// TIA Portal project "s7netcsharp_V16" (V16)

(* hardware
DEVICE "S7300/ET200M station_1"  S7-300 station
   slot 0: "Rail_0"  Rail  6ES7 390-1***0-0AA0
   slot 2: "PLC_1"  CPU 315-2 PN/DP  6ES7 315-2EH14-0AB0  V3.2
      slot 2: "PROFINET interface_1"  PN-IO
         slot 1: "Port_1"  Port
         slot 2: "Port_2"  Port
*)

// ===== PLC "PLC_1"  CPU 315-2 PN/DP =====

VAR_GLOBAL   // PLC tag table "Default tag table"
   "Tag_1" AT %M10.0 : Bool;
   "Tag_2" AT %M10.1 : Bool;
   "Tag_3" AT %M10.2 : Bool;
   "Tag_4" AT %M10.3 : Bool;
   "Tag_5" AT %MW12 : Word;
   "Tag_6" AT %M10.6 : Bool;
   "Tag_7" AT %M10.7 : Bool;
   "Tag_8" AT %MW14 : Word;
   "Tag_9" AT %M11.0 : Bool;
   "Tag_10" AT %M11.1 : Bool;
   "Tag_11" AT %M11.2 : Bool;
   "Tag_12" AT %M11.3 : Bool;
   "Tag_13" AT %M11.4 : Bool;
   "Tag_14" AT %M11.5 : Bool;
   "Tag_15" AT %MW16 : Word;
   "Tag_16" AT %M11.6 : Bool;
   "Tag_17" AT %M20.1 : Bool;
   "Tag_18" AT %M20.2 : Bool;
   "Tag_19" AT %MW22 : Word;
   "Tag_20" AT %M20.4 : Bool;
   "Tag_21" AT %M20.3 : Bool;
   "Tag_22" AT %M20.0 : Bool;
   "Tag_23" AT %M10.4 : Bool;
   "Tag_24" AT %M21.0 : Bool;
   "Tag_25" AT %M21.1 : Bool;
   "AlwaysFalse" AT %M1.0 : Bool;
   "AlwaysTrue" AT %M1.1 : Bool;
   "Tag_26" AT %M0.0 : Bool;
   "Tag_27" AT %M0.1 : Bool;
   "Tag_28" AT %M0.2 : Bool;
   "Tag_29" AT %M0.3 : Bool;
   "Tag_30" AT %M0.4 : Bool;
   "Clock_1Hz" AT %M0.5 : Bool;
   "Time" AT %MD24 : Time;
   "TimeInt" AT %MW28 : Int;
   "pH" AT %MD30 : Real;
END_VAR

DATA_BLOCK "Test"   // DB2
{ S7_Optimized_Access := 'FALSE' }
VERSION : 0.1
   VAR
      Test : Real;
      TestInt : Int;
   END_VAR
BEGIN
END_DATA_BLOCK

// folder: Calculation

DATA_BLOCK "FB_Scale_LI_2"   // DB6
{ S7_Optimized_Access := 'FALSE' }
VERSION : 0.1
// stored: InstanceOfName FB_Scale
"FB_Scale"
BEGIN
END_DATA_BLOCK

DATA_BLOCK "DB_CalculateFlow_FI_1"   // DB13
{ S7_Optimized_Access := 'FALSE' }
VERSION : 0.1
// stored: InstanceOfName FB_CalculateFlow
"FB_CalculateFlow"
BEGIN
END_DATA_BLOCK

DATA_BLOCK "DB_CalculateFlow_FI_2"   // DB14
{ S7_Optimized_Access := 'FALSE' }
VERSION : 0.1
// stored: InstanceOfName FB_CalculateFlow
"FB_CalculateFlow"
BEGIN
END_DATA_BLOCK

DATA_BLOCK "DB_FillingTankT1"   // DB16
{ S7_Optimized_Access := 'FALSE' }
VERSION : 0.1
// stored: InstanceOfName FB_FillingTankT1
"FB_FillingTankT1"
BEGIN
END_DATA_BLOCK

DATA_BLOCK "DB_FillingTankT2"   // DB17
{ S7_Optimized_Access := 'FALSE' }
VERSION : 0.1
// stored: InstanceOfName FB_FillingTankT2
"FB_FillingTankT2"
BEGIN
END_DATA_BLOCK

DATA_BLOCK "FB_Scale_LI_1"   // DB23
{ S7_Optimized_Access := 'FALSE' }
VERSION : 0.1
// stored: InstanceOfName FB_Scale
"FB_Scale"
BEGIN
END_DATA_BLOCK

DATA_BLOCK "DB_PhCalculation"   // DB25
{ S7_Optimized_Access := 'FALSE' }
VERSION : 0.1
// stored: InstanceOfName FB_PhCalculation
"FB_PhCalculation"
BEGIN
END_DATA_BLOCK

DATA_BLOCK "DB_EmptyingCT"   // DB26
{ S7_Optimized_Access := 'FALSE' }
VERSION : 0.1
// stored: InstanceOfName FB_EmptyingCT
"FB_EmptyingCT"
BEGIN
END_DATA_BLOCK

// folder: Measuring Points

DATA_BLOCK "Digital sensors"   // DB7
{ S7_Optimized_Access := 'FALSE' }
VERSION : 0.1
   VAR
      LSHH_T1 : Bool;   // Very high level in Tank 1
      LSLL_T1 : Bool;   // Very low level in Tank 1
      LSHH_T2 : Bool;   // Very high level in Tank 3
      LSLL_T2 : Bool;   // Very low level in Tank 3
      LSH_CT : Bool;   // High level in Chemicals Tank 1
      LSL_CT : Bool;   // Low level in Chemicals Tank 1
   END_VAR
BEGIN
END_DATA_BLOCK

// folder: Measuring Points/Analogs

DATA_BLOCK "DB_Analog_LI_1"   // DB4
{ S7_Optimized_Access := 'FALSE' }
VERSION : 0.1
// stored: InstanceOfName FB_Analog
"FB_Analog"
BEGIN
END_DATA_BLOCK

DATA_BLOCK "DB_Analog_FI_1"   // DB19
{ S7_Optimized_Access := 'FALSE' }
VERSION : 0.1
// stored: InstanceOfName FB_Analog
"FB_Analog"
BEGIN
END_DATA_BLOCK

DATA_BLOCK "DB_Analog_LI_2"   // DB20
{ S7_Optimized_Access := 'FALSE' }
VERSION : 0.1
// stored: InstanceOfName FB_Analog
"FB_Analog"
BEGIN
END_DATA_BLOCK

DATA_BLOCK "DB_Analog_AI_1"   // DB21
{ S7_Optimized_Access := 'FALSE' }
VERSION : 0.1
// stored: InstanceOfName FB_Analog
"FB_Analog"
BEGIN
END_DATA_BLOCK

DATA_BLOCK "DB_Analog_FI_2"   // DB22
{ S7_Optimized_Access := 'FALSE' }
VERSION : 0.1
// stored: InstanceOfName FB_Analog
"FB_Analog"
BEGIN
END_DATA_BLOCK

// folder: Measuring Points/Measuring Transducers

DATA_BLOCK "DB_LI_1"   // DB1
{ S7_Optimized_Access := 'FALSE' }
VERSION : 0.1
// stored: InstanceOfName FB_MeasuringTransducer
"FB_MeasuringTransducer"
BEGIN
END_DATA_BLOCK

DATA_BLOCK "DB_FI_1"   // DB5
{ S7_Optimized_Access := 'FALSE' }
VERSION : 0.1
// stored: InstanceOfName FB_MeasuringTransducer
"FB_MeasuringTransducer"
BEGIN
END_DATA_BLOCK

DATA_BLOCK "DB_LI_2"   // DB28
{ S7_Optimized_Access := 'FALSE' }
VERSION : 0.1
// stored: InstanceOfName FB_MeasuringTransducer
"FB_MeasuringTransducer"
BEGIN
END_DATA_BLOCK

DATA_BLOCK "DB_AI_1"   // DB29
{ S7_Optimized_Access := 'FALSE' }
VERSION : 0.1
// stored: InstanceOfName FB_MeasuringTransducer
"FB_MeasuringTransducer"
BEGIN
END_DATA_BLOCK

DATA_BLOCK "DB_FI_2"   // DB30
{ S7_Optimized_Access := 'FALSE' }
VERSION : 0.1
// stored: InstanceOfName FB_MeasuringTransducer
"FB_MeasuringTransducer"
BEGIN
END_DATA_BLOCK

// folder: Program files

DATA_BLOCK "DB_FILL_T1"   // DB12
{ S7_Optimized_Access := 'FALSE' }
VERSION : 0.1
   VAR
      START : Bool;   // Start signal from SCADA
      SET_START : Bool;   // Set start signal
      STOP : Bool;   // Stop signal from SCADA
      SET_STOP : Bool;   // Set stop signal
      UV_1_OPEN : Bool;   // Open valve UV_1
      STATE : Int;   // 0 - Stop, 1 - Filling T1, 2 - No conditions to run
   END_VAR
BEGIN
END_DATA_BLOCK

DATA_BLOCK "DB_TRANSFER_TO_T2"   // DB18
{ S7_Optimized_Access := 'FALSE' }
VERSION : 0.1
   VAR
      START : Bool;   // Start signal from SCADA
      SET_START : Bool;   // Set start signal
      STOP : Bool;   // Stop signal from SCADA
      SET_STOP : Bool;   // Set stop signal
      Spare : Bool;   // Spare
      P1_START : Bool;   // Start signal for Pump P1
      UV_2_OPEN : Bool;   // Open valve UV_2
      SetPhVal : Bool;   // Set random ph value signal
      LI_2_SP : Real := 7000.0;   // Setpoint for Tank T2 filling level
      AI_1_SetVal : Real;   // Random Value of Ph in Tank T3
      STATE : Int;   // 0 - Stop, 1 - Transfer to T2, 2 - Adding chemicals, 3 - No conditions to run
      P1_SP : Real;   // Pump P1 Speed Setpoint
   END_VAR
BEGIN
END_DATA_BLOCK

DATA_BLOCK "DB_DOSE_CHEMICALS"   // DB24
{ S7_Optimized_Access := 'FALSE' }
VERSION : 0.1
   VAR
      START : Bool;   // Start signal from SCADA
      SET_START : Bool;   // Set start signal
      STOP : Bool;   // Stop signal from SCADA
      SET_STOP : Bool;   // Set stop signal
      P3_START : Bool;
      STATE : Int;   // 0 - Stop, 1 - Adding Chemicals, 2 - No conditions to run
   END_VAR
BEGIN
END_DATA_BLOCK

DATA_BLOCK "DB_EMPTYING_T2"   // DB27
{ S7_Optimized_Access := 'FALSE' }
VERSION : 0.1
   VAR
      START : Bool;   // Start signal from SCADA
      SET_START : Bool;   // Set start signal
      STOP : Bool;   // Stop signal from SCADA
      SET_STOP : Bool;   // Set stop signal
      P2_START : Bool;   // Start signal for Pump P2
      Spare : Bool;
      Spare_1 : Bool;
      Spare_2 : Bool;
      State : Int;   // 0 - stop, 1 - Emptying, 3 - No conditions to run
      P2_SP : Real;   // Pump P2 Speed Setpoint
   END_VAR
BEGIN
END_DATA_BLOCK

// folder: Pumps

DATA_BLOCK "DB_Pump_P1"   // DB8
{ S7_Optimized_Access := 'FALSE' }
VERSION : 0.1
// stored: InstanceOfName FB_MotorControl
"FB_MotorControl"
BEGIN
END_DATA_BLOCK

DATA_BLOCK "DB_Pump_P2"   // DB9
{ S7_Optimized_Access := 'FALSE' }
VERSION : 0.1
// stored: InstanceOfName FB_MotorControl
"FB_MotorControl"
BEGIN
END_DATA_BLOCK

DATA_BLOCK "DB_Pump_P3"   // DB15
{ S7_Optimized_Access := 'FALSE' }
VERSION : 0.1
// stored: InstanceOfName FB_MotorControl
"FB_MotorControl"
BEGIN
END_DATA_BLOCK

// folder: Valves

DATA_BLOCK "DB_UV_1"   // DB10
{ S7_Optimized_Access := 'FALSE' }
VERSION : 0.1
// stored: InstanceOfName FB_Valve
"FB_Valve"
BEGIN
END_DATA_BLOCK

DATA_BLOCK "DB_UV_2"   // DB11
{ S7_Optimized_Access := 'FALSE' }
VERSION : 0.1
// stored: InstanceOfName FB_Valve
"FB_Valve"
BEGIN
END_DATA_BLOCK

// folder: (top level)

FUNCTION_BLOCK "FB_MeasuringTransducer"   // FB1, SCL
{ S7_Optimized_Access := 'FALSE' }
VERSION : 0.1
   VAR_INPUT
      X : Real;   // Input value (Final respond transducer value
      T1 : Time;   // Main constant transducer value
      T2 : Time;   // Second constant transducer value
      Ts : Time;   // Sampling time
      K : Real;   // Gain
   END_VAR
   VAR_OUTPUT
      Y : Real;   // Output value
   END_VAR
   VAR
      Yn1 : Real;
      Yn2 : Real;
      T_Sampling : Real;
      T1_Temp : Real;
      T2_Temp : Real;
   END_VAR
BEGIN
   // Input time conversion
   #T_Sampling := (DINT_TO_REAL(TIME_TO_DINT(#Ts))) / 1000.0;
   #T1_Temp := (DINT_TO_REAL(TIME_TO_DINT(#T1))) / 1000.0;
   #T2_Temp := (DINT_TO_REAL(TIME_TO_DINT(#T2))) / 1000.0;

   // ***************************************************
   // Second order measuring transducer Euler's equation
   // For more details go to Readme.txt file
   // ***************************************************

   #Y := ((#K * (#T_Sampling * #T_Sampling) * #X) + ((#T_Sampling
   * #T1_Temp + 2 * #T1_Temp * #T2_Temp + #T_Sampling * #T2_Temp) *
   #Yn1) - ((#T1_Temp * #T2_Temp) * #Yn2)) / ((#T_Sampling *
   #T_Sampling) + #T_Sampling * #T2_Temp + #T_Sampling * #T1_Temp +
   #T1_Temp * #T2_Temp);

   #Yn2 := #Yn1;
   #Yn1 := #Y;
END_FUNCTION_BLOCK

FUNCTION_BLOCK "FB_MotorControl"   // FB2, SCL
{ S7_Optimized_Access := 'FALSE' }
VERSION : 0.1
   VAR_INPUT
      START : Bool;   // Start in auto mode
      BLOCKADE : Bool;
      TRIGGER : Bool;   // Time trigger for running time
      SP_IN : Real;   // Setpoint [%]
   END_VAR
   VAR_OUTPUT
      RUNNING : Bool;
      FAULT : Bool;
      ERROR_CODE : Int;
      STATE : Int;   // 0 - stop, 1 - starting up, 2 - run, 3 - stopping, 4 - blockade active, 5 - fault
      PV : Real;
   END_VAR
   VAR
      MODE : Bool := false;   // 0 - auto, 1 - manual
      SCADA : Struct   // Signals from/to Scada
         START : Bool;   // Start signal from Scada
         STOP : Bool;   // Stop signal from Scada
         AUTO : Bool := false;   // Auto mode signal from Scada
         MANUAL : Bool;   // Manual mode signal from Scada
         BLOCKADE : Bool;   // 0 - blockade unactive, 1 - blockade active
         FAULT : Bool;   // Motor fault info to Scada
         RUN_H : Int;   // Running time - hours
         RUN_MIN : Int;   // Running time - minutes
         RUN_S : Int;   // Running time - seconds
         RESET_TIME : Bool;   // Reset running time
         MODE : Bool;   // 0 - auto, 1 - manual (Scada)
         STATE : Int;   // 0 - stop, 1 - starting up, 2 - running, 3 - stopping, 4 - blockade active, 5 - fault
         SP : Real;   // Setpoint value [%]
         PV : Real;
      END_STRUCT;
      Yn1 : Real;
      Yn2 : Real;
      T_Sampling : Real;
      T1_Temp : Real;
      T2_Temp : Real;
      SP : Real;
      SignalOld : Bool;
   END_VAR
   VAR_TEMP
      Edge : Bool;
   END_VAR
   VAR CONSTANT
      T1 : Time := T#1s;   // Main constant transducer value
      T2 : Time := T#500ms;   // Second constant transducer value
      Ts : Time := T#100ms;   // Sampling time
      K : Real := 1.0;   // Gain
   END_VAR
BEGIN
   #SCADA.BLOCKADE := #BLOCKADE;
   #SCADA.FAULT := #FAULT;
   #SCADA.STATE := #STATE;

   // Input time conversion
   #T_Sampling := (DINT_TO_REAL(TIME_TO_DINT(#Ts))) / 1000.0;
   #T1_Temp := (DINT_TO_REAL(TIME_TO_DINT(#T1))) / 1000.0;
   #T2_Temp := (DINT_TO_REAL(TIME_TO_DINT(#T2))) / 1000.0;

   // Positive edge detection
   #Edge := #TRIGGER AND NOT #SignalOld;
   #SignalOld := #TRIGGER;

   // Blockade
   IF (#BLOCKADE) THEN
       #ERROR_CODE := 1;
       #START := FALSE;
       #SCADA.START := FALSE;
       #SCADA.STOP := TRUE;
       #RUNNING := FALSE;
       #FAULT := TRUE;
       #SP := 0;
       #STATE := 4;
   END_IF;

   // Manual and auto mode set
   IF (#SCADA.MANUAL) THEN
       #MODE := TRUE;
   ELSIF (#SCADA.AUTO) THEN
       #MODE := FALSE;
   END_IF;

   // Main program
   IF (#BLOCKADE = FALSE) THEN
       #FAULT := FALSE;
       IF (#MODE = FALSE AND #START = TRUE) THEN
           #RUNNING := TRUE;
           #SP := #SP_IN;

           //Status change - starting up/run
           IF (#SP * 0.90 > #PV) THEN
               #STATE := 1;
           ELSIF (#SP * 0.90 < #PV) THEN
               #STATE := 2;
           END_IF;

       ELSIF (#MODE = FALSE AND #START = FALSE) THEN
           #RUNNING := FALSE;
           #SP := 0.0;
           //Status change - stopping/stop
           IF (0.05 < #PV) THEN
               #STATE := 3;
           ELSIF (0.05 > #PV) THEN
               #STATE := 4;
           END_IF;

       ELSIF(#MODE = TRUE AND #SCADA.START = TRUE) THEN
           #RUNNING := TRUE;
           #SP := #SCADA.SP;
           //Status change - starting up/runn
           IF (#SP * 0.90 > #PV) THEN
               #STATE := 1;
           ELSIF (#SP * 0.90 < #PV) THEN
               #STATE := 2;
           END_IF;

       ELSIF (#MODE = TRUE AND #SCADA.START = FALSE) THEN
           #RUNNING := FALSE;
           #SP := 0.0;
           //Status change - stopping/stop
           IF (0.05 < #PV) THEN
               #STATE := 3;
           ELSIF (0.05 > #PV) THEN
               #STATE := 4;
           END_IF;

       END_IF;
   END_IF;

   // Euler's second order equation for simulate acceleration and slowing down  
   #PV := ((#K * (#T_Sampling * #T_Sampling) * #SP) + ((#T_Sampling
   * #T1_Temp + 2 * #T1_Temp * #T2_Temp + #T_Sampling * #T2_Temp) *
   #Yn1) - ((#T1_Temp * #T2_Temp) * #Yn2)) / ((#T_Sampling *
   #T_Sampling) + #T_Sampling * #T2_Temp + #T_Sampling * #T1_Temp +
   #T1_Temp * #T2_Temp);
   #Yn2 := #Yn1;
   #Yn1 := #PV;

   // Running time
   IF (#RUNNING AND #Edge) THEN
       #SCADA.RUN_S := #SCADA.RUN_S+1;
       IF (#SCADA.RUN_S = 60) THEN
           #SCADA.RUN_S := 0;
           #SCADA.RUN_MIN := #SCADA.RUN_MIN+1;
       END_IF;

       IF (#SCADA.RUN_MIN = 60) THEN
           #SCADA.RUN_MIN := 0;
           #SCADA.RUN_H := #SCADA.RUN_H+1;
       END_IF;

   END_IF;

   // Reset running time
   IF (#SCADA.RESET_TIME) THEN
       #SCADA.RUN_S := 0;
       #SCADA.RUN_MIN := 0;
       #SCADA.RUN_H := 0;
   END_IF;

   // 
   // STATUS CODES
   // 1: Blockade active
   //
END_FUNCTION_BLOCK

FUNCTION_BLOCK "FB_Valve"   // FB3, SCL
{ S7_Optimized_Access := 'FALSE' }
VERSION : 0.1
   VAR_INPUT
      "OPEN/CLOSE" : Bool;   // 0 - Close, 1 - Open
      BLOCKADE : Bool;
      DETECT_TIME : Int;   // Time of Inefficient open / close detection error [s]
   END_VAR
   VAR_OUTPUT
      STATE : Int;   // 0 - Closed, 1 - Closing, 2 - Open, 3 - Opening, 4 - Fault
      FAULT : Bool;
      ERROR_CODE : Int;
      OUT : Bool;   // 0 - Close, 1 - Open
      CLOSE_LIMIT : Bool;   // Closing limit
      OPEN_LIMIT : Bool;   // Opening limit
   END_VAR
   VAR
      SCADA : Struct
         OPEN : Bool;   // Open valve singal from scada
         CLOSE : Bool;   // Close valve singal from scada
         AUTO : Bool;   // Auto mode signal from scada
         MANUAL : Bool;   // Manual mode signal from scada
         FAULT : Bool;   // Valve fault
         BLOCKADE : Bool;   // 1 - Blockade active
         AM : Bool;   // 0 - Auto, 1 - Manual
         OPEN_CLOSE : Bool;   // 0 - Closing, 1 - Opening
         STATE : Int;   // 0 - Closed, 1 - Closing, 2 - Open, 3 - Opening
      END_STRUCT;
      SignalOld : Bool;
      OpenDetTime : Int;
      CloseDetTime : Int;
   END_VAR
   VAR_TEMP
      EDGE : Bool;
   END_VAR
BEGIN
   #SCADA.STATE := #STATE;
   #SCADA.FAULT := #FAULT;
   #SCADA.BLOCKADE := #BLOCKADE;
   // Positive edge detection
   #EDGE := "Clock_1Hz" AND NOT #SignalOld;
   #SignalOld := "Clock_1Hz";

   // Open / Close from scada
   IF (#SCADA.OPEN) THEN
       #SCADA.OPEN_CLOSE := TRUE;
       #SCADA.OPEN := FALSE;
   ELSIF (#SCADA.CLOSE) THEN
       #SCADA.OPEN_CLOSE := FALSE;
       #SCADA.CLOSE := FALSE;
   END_IF;

   // Auto / Manual from scada
   IF (#SCADA.MANUAL) THEN
       #SCADA.AM := TRUE;
       #SCADA.MANUAL := FALSE;
   ELSIF (#SCADA.AUTO) THEN
       #SCADA.AM := FALSE;
       #SCADA.AUTO := FALSE;
   END_IF;

   IF (#BLOCKADE) THEN
       #FAULT := TRUE;
       #OUT := FALSE;
       #ERROR_CODE := 1;
       #OpenDetTime := 0;

       //Close valve when blockade is on
       IF (#EDGE AND #CloseDetTime <> #DETECT_TIME) THEN
           #CloseDetTime := #CloseDetTime + 1;
           #STATE := 1;

           IF (#CloseDetTime = #DETECT_TIME) THEN
               #OUT := TRUE;
               #STATE := 0;
               #OPEN_LIMIT := FALSE;
               #CLOSE_LIMIT := TRUE;
           END_IF;

       END_IF;

   ELSIF (#BLOCKADE = FALSE) THEN
       #FAULT := FALSE;
       // Manual Mode
       IF (#SCADA.AM) THEN
           // Opening the valve
           IF (#SCADA.OPEN_CLOSE) THEN
               #CloseDetTime := 0;
               IF (#EDGE AND #OpenDetTime <> #DETECT_TIME) THEN
                   #OpenDetTime := #OpenDetTime + 1;
                   #STATE := 3;

                   IF (#OpenDetTime = #DETECT_TIME) THEN
                       #OUT := TRUE;
                       #STATE := 2;
                       #CLOSE_LIMIT := FALSE;
                       #OPEN_LIMIT := TRUE;
                   END_IF;

               END_IF;
           // Closing valve
           ELSIF (#SCADA.OPEN_CLOSE=FALSE) THEN
               #OpenDetTime := 0;
               IF (#EDGE AND #CloseDetTime <> #DETECT_TIME) THEN
                   #CloseDetTime := #CloseDetTime + 1;
                   #STATE := 1;

                   IF (#CloseDetTime = #DETECT_TIME) THEN
                       #OUT := TRUE;
                       #STATE := 0;
                       #OPEN_LIMIT := FALSE;
                       #CLOSE_LIMIT := TRUE;
                   END_IF;

               END_IF;
           END_IF;
       // Automatic mode    
       ELSIF (#SCADA.AM = FALSE) THEN
           // Opening the valve
           IF (#"OPEN/CLOSE") THEN
               #CloseDetTime := 0;
               IF (#EDGE AND #OpenDetTime <> #DETECT_TIME) THEN
                   #OpenDetTime := #OpenDetTime + 1;
                   #STATE := 3;

                   IF (#OpenDetTime = #DETECT_TIME) THEN
                       #OUT := TRUE;
                       #STATE := 2;
                       #CLOSE_LIMIT := FALSE;
                       #OPEN_LIMIT := TRUE;
                   END_IF;

               END_IF;
           // Closing valve    
           ELSIF (#"OPEN/CLOSE" = FALSE) THEN
               #OpenDetTime := 0;
               IF (#EDGE AND #CloseDetTime <> #DETECT_TIME) THEN
                   #CloseDetTime := #CloseDetTime + 1;
                   #STATE := 1;

                   IF (#CloseDetTime = #DETECT_TIME) THEN
                       #OUT := TRUE;
                       #STATE := 0;
                       #OPEN_LIMIT := FALSE;
                       #CLOSE_LIMIT := TRUE;
                   END_IF;

               END_IF;
           END_IF;

       END_IF;

   END_IF;
END_FUNCTION_BLOCK

FUNCTION_BLOCK "FB_Scale"   // FB7, SCL
{ S7_Optimized_Access := 'FALSE' }
VERSION : 0.1
   VAR_INPUT
      VALUE : Real;
      HI_RANGE : Real;
   END_VAR
   VAR_OUTPUT
      OUT_PRC : Real;
   END_VAR
BEGIN
   // Scale input value to percent

   #OUT_PRC := DINT_TO_REAL(ROUND(((#VALUE * 100.0) / #HI_RANGE) *100.0))/100.0;
END_FUNCTION_BLOCK

FUNCTION_BLOCK "FB_RandomPhGenerator"   // FB10, SCL
{ S7_Optimized_Access := 'FALSE' }
VERSION : 0.1
   VAR_INPUT
      LowRange : Real;   // Minimum input ph value ( 0 - min)
      HghRange : Real;   // Maximum input ph value (10 - max)
   END_VAR
   VAR_OUTPUT
      Value : Real;
      Error : Bool;   // Wrong input value (1-10ph)
   END_VAR
   VAR
      "Time" : Date_And_Time;
      Seconds : Int;
   END_VAR
   VAR_TEMP
      RetVal : Int;
   END_VAR
BEGIN
   #RetVal:=RD_SYS_T(OUT => #Time);
END_FUNCTION_BLOCK

FUNCTION_BLOCK "FB_Analog"   // FB11, SCL
{ S7_Optimized_Access := 'FALSE' }
VERSION : 0.1
   VAR_INPUT
      Value : Real;   // Measured Value
      HHI : Bool;   // Very high level of measured value (Alarm)
      HI : Bool;   // High level of measured value (Warning)
      LO : Bool;   // Low level of measured value (Warning)
      LLO : Bool;   // Very low level of measured value (Alarm)
      HHI_SP : Real;   // Setpoint for very high level detection
      HI_SP : Real;   // Setpoint for vhigh level detection
      LO_SP : Real;   // Setpoint for low level detection
      LLO_SP : Real;   // Setpoint for very low level detection
   END_VAR
   VAR_OUTPUT
      HHI_ALARM : Bool;
      HI_WARN : Bool;
      LO_WARN : Bool;
      LLO_ALARM : Bool;
   END_VAR
BEGIN
   // Very high level detection
   IF (#HHI) THEN
       IF (#Value >= #HHI_SP) THEN
           #HHI_ALARM := TRUE;
       ELSIF (#Value < #HHI_SP) THEN
           #HHI_ALARM := FALSE;
       END_IF;
   END_IF;
   // High level detection
   IF (#HI) THEN
       IF (#Value >= #HI_SP) THEN
           #HI_WARN := TRUE;
       ELSIF (#Value < #HI_SP) THEN
           #HI_WARN := FALSE;
       END_IF;
   END_IF;
   // Low level detection
   IF (#LO) THEN
       IF (#Value >= #LO_SP) THEN
           #LO_WARN := TRUE;
       ELSIF (#Value < #LO_SP) THEN
           #LO_WARN := FALSE;
       END_IF;
   END_IF;
   // Very low level detection
   IF (#LLO) THEN
       IF (#Value >= #LLO_SP) THEN
           #LLO_ALARM := TRUE;
       ELSIF (#Value < #LLO_SP) THEN
           #LLO_ALARM := FALSE;
       END_IF;
   END_IF;
END_FUNCTION_BLOCK

FUNCTION "FC_RandomPhGenerator" : Void   // FC1, SCL
{ S7_Optimized_Access := 'FALSE' }
VERSION : 0.1
   VAR_INPUT
      Value : Int;
      LowRange : Real;   // Lowest ph Value
      HighRange : Real;   // Highest ph Value
   END_VAR
   VAR_OUTPUT
      pH : Real;
   END_VAR
   VAR_TEMP
      TemVal : Real;
      TempPh : Real;
   END_VAR
BEGIN
   IF (#Value > 0) THEN
       #TemVal := INT_TO_REAL(#Value);
   ELSIF (#Value < 0) THEN
       #TemVal := INT_TO_REAL(#Value * -1);
   END_IF;
   #TempPh := ((#TemVal/100)/5.46)/10.0;

   IF (#TempPh < #LowRange) THEN
       #pH := #LowRange;
   ELSIF (#TempPh > #HighRange) THEN
       #pH := #HighRange;
   ELSE
       #pH := #TempPh;
   END_IF;
END_FUNCTION

FUNCTION "FC_Limits" : Void   // FC8, LAD
{ S7_Optimized_Access := 'FALSE' }
VERSION : 0.1
BEGIN

REGION Network 1: LSHH T1 - Limit
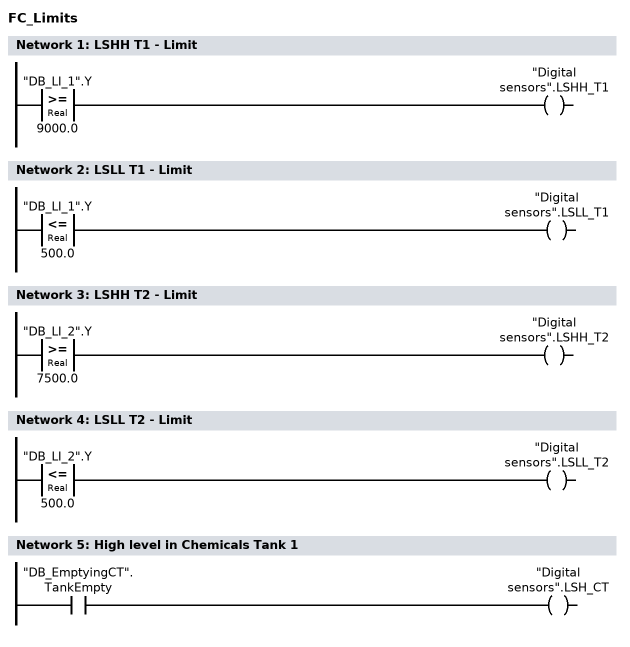
   RUNG wire#powerrail
      { S7_Templates := "SrcType := Real" } GE_Contact(in1 := "DB_LI_1".Y, in2 := 9000.0)
      Coil( "Digital sensors".LSHH_T1 )
   END_RUNG
   // the same network as SCL:
   "Digital sensors".LSHH_T1 := "DB_LI_1".Y >= 9000.0;
END_REGION

REGION Network 2: LSLL T1 - Limit
   RUNG wire#powerrail
      { S7_Templates := "SrcType := Real" } LE_Contact(in1 := "DB_LI_1".Y, in2 := 500.0)
      Coil( "Digital sensors".LSLL_T1 )
   END_RUNG
   // the same network as SCL:
   "Digital sensors".LSLL_T1 := "DB_LI_1".Y <= 500.0;
END_REGION

REGION Network 3: LSHH T2 - Limit
   RUNG wire#powerrail
      { S7_Templates := "SrcType := Real" } GE_Contact(in1 := "DB_LI_2".Y, in2 := 7500.0)
      Coil( "Digital sensors".LSHH_T2 )
   END_RUNG
   // the same network as SCL:
   "Digital sensors".LSHH_T2 := "DB_LI_2".Y >= 7500.0;
END_REGION

REGION Network 4: LSLL T2 - Limit
   RUNG wire#powerrail
      { S7_Templates := "SrcType := Real" } LE_Contact(in1 := "DB_LI_2".Y, in2 := 500.0)
      Coil( "Digital sensors".LSLL_T2 )
   END_RUNG
   // the same network as SCL:
   "Digital sensors".LSLL_T2 := "DB_LI_2".Y <= 500.0;
END_REGION

REGION Network 5: High level in Chemicals Tank 1
   RUNG wire#powerrail
      Contact( "DB_EmptyingCT".TankEmpty )
      Coil( "Digital sensors".LSH_CT )
   END_RUNG
   // the same network as SCL:
   "Digital sensors".LSH_CT := "DB_EmptyingCT".TankEmpty;
END_REGION
END_FUNCTION

ORGANIZATION_BLOCK "Main"   // OB1, LAD
TITLE = "Main Program Sweep (Cycle)"
{ S7_Optimized_Access := 'FALSE' }
VERSION : 0.1
   VAR_TEMP
      OB1_EV_CLASS : Byte;   // Bits 0-3 = 1 (Coming event), Bits 4-7 = 1 (Event class 1)
      OB1_SCAN_1 : Byte;   // 1 (Cold restart scan 1 of OB 1), 3 (Scan 2-n of OB 1)
      OB1_PRIORITY : Byte;   // Priority of OB Execution
      OB1_OB_NUMBR : Byte;   // 1 (Organization block 1, OB1)
      OB1_RESERVED_1 : Byte;   // Reserved for system
      OB1_RESERVED_2 : Byte;   // Reserved for system
      OB1_PREV_CYCLE : Int;   // Cycle time of previous OB1 scan (milliseconds)
      OB1_MIN_CYCLE : Int;   // Minimum cycle time of OB1 (milliseconds)
      OB1_MAX_CYCLE : Int;   // Maximum cycle time of OB1 (milliseconds)
      OB1_DATE_TIME : Date_And_Time;   // Date and time OB1 started
   END_VAR
BEGIN

REGION Network 1: Always False / True
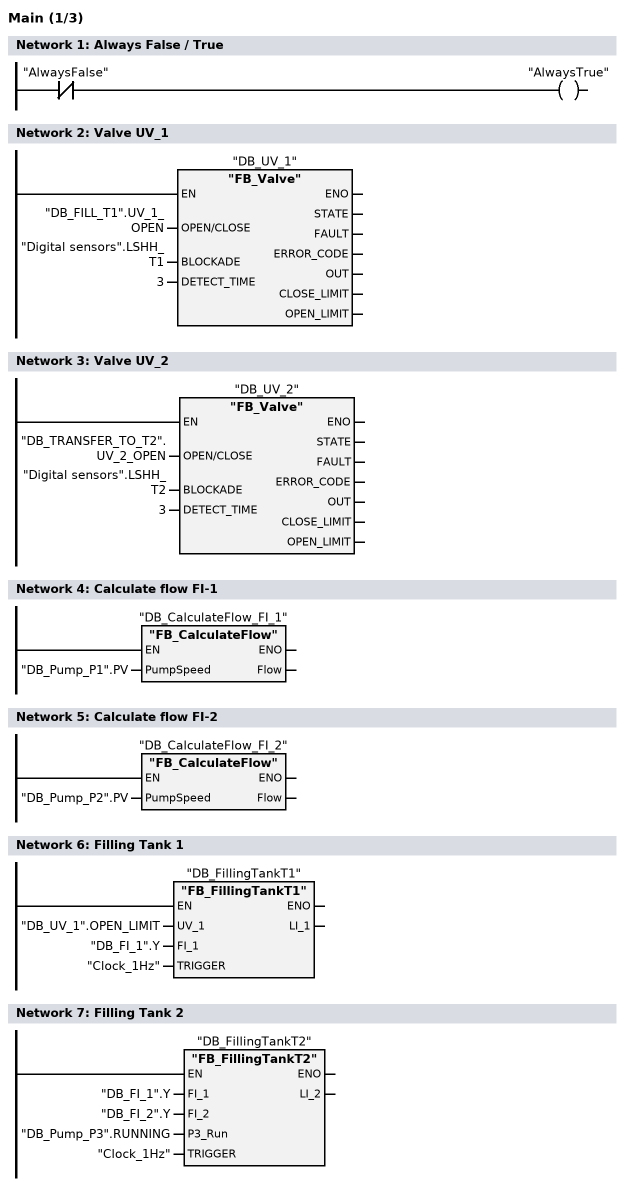
   RUNG wire#powerrail
      I_Contact( "AlwaysFalse" )
      Coil( "AlwaysTrue" )
   END_RUNG
   // the same network as SCL:
   "AlwaysTrue" := NOT "AlwaysFalse";
END_REGION

REGION Network 2: Valve UV_1
   RUNG wire#powerrail
      "DB_UV_1"("OPEN/CLOSE" := "DB_FILL_T1".UV_1_OPEN, BLOCKADE := "Digital sensors".LSHH_T1, DETECT_TIME := 3, STATE =>, FAULT =>, ERROR_CODE =>, OUT =>, CLOSE_LIMIT =>, OPEN_LIMIT =>)
   END_RUNG
   // the same network as SCL:
   "DB_UV_1"("OPEN/CLOSE" := "DB_FILL_T1".UV_1_OPEN, BLOCKADE := "Digital sensors".LSHH_T1, DETECT_TIME := 3);   // "FB_Valve"
END_REGION

REGION Network 3: Valve UV_2
   RUNG wire#powerrail
      "DB_UV_2"("OPEN/CLOSE" := "DB_TRANSFER_TO_T2".UV_2_OPEN, BLOCKADE := "Digital sensors".LSHH_T2, DETECT_TIME := 3, STATE =>, FAULT =>, ERROR_CODE =>, OUT =>, CLOSE_LIMIT =>, OPEN_LIMIT =>)
   END_RUNG
   // the same network as SCL:
   "DB_UV_2"("OPEN/CLOSE" := "DB_TRANSFER_TO_T2".UV_2_OPEN,   // "FB_Valve"
             BLOCKADE := "Digital sensors".LSHH_T2,
             DETECT_TIME := 3);
END_REGION

REGION Network 4: Calculate flow FI-1
   RUNG wire#powerrail
      "DB_CalculateFlow_FI_1"(PumpSpeed := "DB_Pump_P1".PV, Flow =>)
   END_RUNG
   // the same network as SCL:
   "DB_CalculateFlow_FI_1"(PumpSpeed := "DB_Pump_P1".PV);   // "FB_CalculateFlow"
END_REGION

REGION Network 5: Calculate flow FI-2
   RUNG wire#powerrail
      "DB_CalculateFlow_FI_2"(PumpSpeed := "DB_Pump_P2".PV, Flow =>)
   END_RUNG
   // the same network as SCL:
   "DB_CalculateFlow_FI_2"(PumpSpeed := "DB_Pump_P2".PV);   // "FB_CalculateFlow"
END_REGION

REGION Network 6: Filling Tank 1
   RUNG wire#powerrail
      "DB_FillingTankT1"(UV_1 := "DB_UV_1".OPEN_LIMIT, FI_1 := "DB_FI_1".Y, TRIGGER := "Clock_1Hz", LI_1 =>)
   END_RUNG
   // the same network as SCL:
   "DB_FillingTankT1"(UV_1 := "DB_UV_1".OPEN_LIMIT, FI_1 := "DB_FI_1".Y, TRIGGER := "Clock_1Hz");   // "FB_FillingTankT1"
END_REGION

REGION Network 7: Filling Tank 2
   RUNG wire#powerrail
      "DB_FillingTankT2"(FI_1 := "DB_FI_1".Y, FI_2 := "DB_FI_2".Y, P3_Run := "DB_Pump_P3".RUNNING, TRIGGER := "Clock_1Hz", LI_2 =>)
   END_RUNG
   // the same network as SCL:
   "DB_FillingTankT2"(FI_1 := "DB_FI_1".Y,   // "FB_FillingTankT2"
                      FI_2 := "DB_FI_2".Y,
                      P3_Run := "DB_Pump_P3".RUNNING,
                      TRIGGER := "Clock_1Hz");
END_REGION

REGION Network 8: PhCalculation
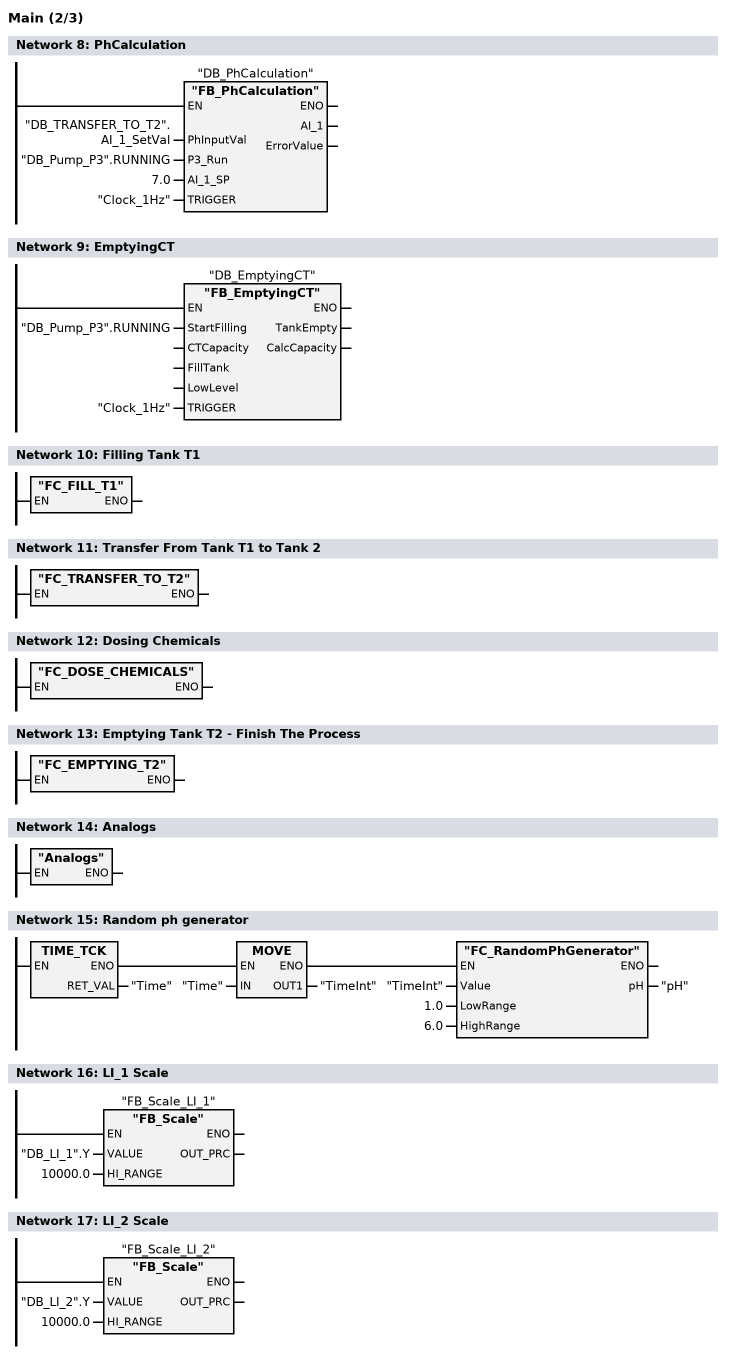
   RUNG wire#powerrail
      "DB_PhCalculation"(PhInputVal := "DB_TRANSFER_TO_T2".AI_1_SetVal, P3_Run := "DB_Pump_P3".RUNNING, AI_1_SP := 7.0, TRIGGER := "Clock_1Hz", AI_1 =>, ErrorValue =>)
   END_RUNG
   // the same network as SCL:
   "DB_PhCalculation"(PhInputVal := "DB_TRANSFER_TO_T2".AI_1_SetVal,   // "FB_PhCalculation"
                      P3_Run := "DB_Pump_P3".RUNNING,
                      AI_1_SP := 7.0,
                      TRIGGER := "Clock_1Hz");
END_REGION

REGION Network 9: EmptyingCT
   RUNG wire#powerrail
      "DB_EmptyingCT"(StartFilling := "DB_Pump_P3".RUNNING, CTCapacity :=, FillTank :=, LowLevel :=, TRIGGER := "Clock_1Hz", TankEmpty =>, CalcCapacity =>)
   END_RUNG
   // the same network as SCL:
   "DB_EmptyingCT"(StartFilling := "DB_Pump_P3".RUNNING, TRIGGER := "Clock_1Hz");   // "FB_EmptyingCT"
END_REGION

REGION Network 10: Filling Tank T1
   RUNG wire#powerrail
      "FC_FILL_T1"()
   END_RUNG
   // the same network as SCL:
   "FC_FILL_T1"();
END_REGION

REGION Network 11: Transfer From Tank T1 to Tank 2
   RUNG wire#powerrail
      "FC_TRANSFER_TO_T2"()
   END_RUNG
   // the same network as SCL:
   "FC_TRANSFER_TO_T2"();
END_REGION

REGION Network 12: Dosing Chemicals
   RUNG wire#powerrail
      "FC_DOSE_CHEMICALS"()
   END_RUNG
   // the same network as SCL:
   "FC_DOSE_CHEMICALS"();
END_REGION

REGION Network 13: Emptying Tank T2 - Finish The Process
   RUNG wire#powerrail
      "FC_EMPTYING_T2"()
   END_RUNG
   // the same network as SCL:
   "FC_EMPTYING_T2"();
END_REGION

REGION Network 14: Analogs
   RUNG wire#powerrail
      "Analogs"()
   END_RUNG
   // the same network as SCL:
   "Analogs"();
END_REGION

REGION Network 15: Random ph generator
   // ENO of a box is taken as its EN; it also drops when the box reports an error
   "Time" := TIME_TCK();
   "TimeInt" := "Time";
   "FC_RandomPhGenerator"(Value := "TimeInt", LowRange := 1.0, HighRange := 6.0, pH => "pH");
END_REGION

REGION Network 16: LI_1 Scale
   RUNG wire#powerrail
      "FB_Scale_LI_1"(VALUE := "DB_LI_1".Y, HI_RANGE := 10000.0, OUT_PRC =>)
   END_RUNG
   // the same network as SCL:
   "FB_Scale_LI_1"(VALUE := "DB_LI_1".Y, HI_RANGE := 10000.0);   // "FB_Scale"
END_REGION

REGION Network 17: LI_2 Scale
   RUNG wire#powerrail
      "FB_Scale_LI_2"(VALUE := "DB_LI_2".Y, HI_RANGE := 10000.0, OUT_PRC =>)
   END_RUNG
   // the same network as SCL:
   "FB_Scale_LI_2"(VALUE := "DB_LI_2".Y, HI_RANGE := 10000.0);   // "FB_Scale"
END_REGION

REGION Network 18: Limits
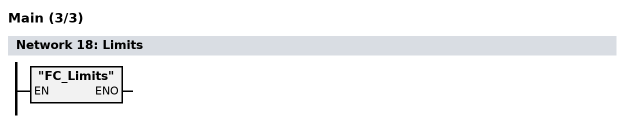
   RUNG wire#powerrail
      "FC_Limits"()
   END_RUNG
   // the same network as SCL:
   "FC_Limits"();
END_REGION
END_ORGANIZATION_BLOCK

ORGANIZATION_BLOCK "CYC_INT5"   // OB35, FBD
TITLE = "Cyclic Interrupt"
{ S7_Optimized_Access := 'FALSE' }
VERSION : 0.1
   VAR_TEMP
      OB35_EV_CLASS : Byte;   // Bits 0-3 = 1 (Coming event), Bits 4-7 = 1 (Event class 1)
      OB35_STRT_INF : Byte;   // 16#36 (OB 35 has started)
      OB35_PRIORITY : Byte;   // Priority of OB Execution
      OB35_OB_NUMBR : Byte;   // 35 (Organization block 35, OB35)
      OB35_RESERVED_1 : Byte;   // Reserved for system
      OB35_RESERVED_2 : Byte;   // Reserved for system
      OB35_PHASE_OFFSET : Word;   // Phase offset (msec)
      OB35_RESERVED_3 : Int;   // Reserved for system
      OB35_EXC_FREQ : Int;   // Frequency of execution (msec)
      OB35_DATE_TIME : Date_And_Time;   // Date and time OB35 started
   END_VAR
BEGIN

REGION Network 1: Measuring Transducers
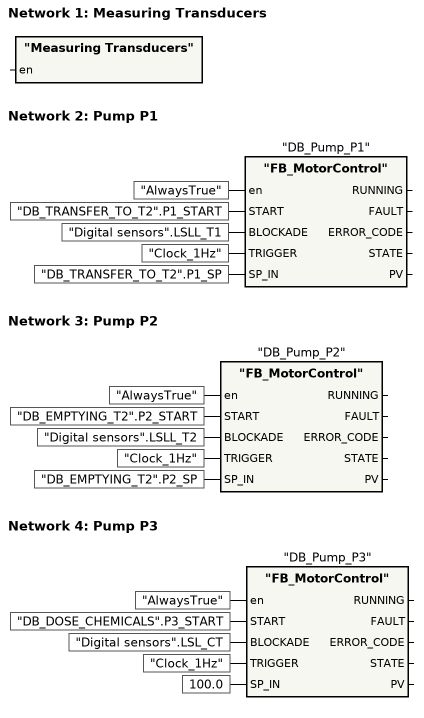
   "Measuring Transducers"();
END_REGION

REGION Network 2: Pump P1
   IF "AlwaysTrue" THEN
       "DB_Pump_P1"(START := "DB_TRANSFER_TO_T2".P1_START,   // "FB_MotorControl"
                    BLOCKADE := "Digital sensors".LSLL_T1,
                    TRIGGER := "Clock_1Hz",
                    SP_IN := "DB_TRANSFER_TO_T2".P1_SP);
   END_IF;
END_REGION

REGION Network 3: Pump P2
   IF "AlwaysTrue" THEN
       "DB_Pump_P2"(START := "DB_EMPTYING_T2".P2_START,   // "FB_MotorControl"
                    BLOCKADE := "Digital sensors".LSLL_T2,
                    TRIGGER := "Clock_1Hz",
                    SP_IN := "DB_EMPTYING_T2".P2_SP);
   END_IF;
END_REGION

REGION Network 4: Pump P3
   IF "AlwaysTrue" THEN
       "DB_Pump_P3"(START := "DB_DOSE_CHEMICALS".P3_START,   // "FB_MotorControl"
                    BLOCKADE := "Digital sensors".LSL_CT,
                    TRIGGER := "Clock_1Hz",
                    SP_IN := 100.0);
   END_IF;
END_REGION
END_ORGANIZATION_BLOCK

ORGANIZATION_BLOCK "CYCL_FLT"   // OB80, LAD
TITLE = "Cycle Time Fault"
{ S7_Optimized_Access := 'FALSE' }
VERSION : 0.1
   VAR_TEMP
      OB80_EV_CLASS : Byte;   // 16#35, Event class 3, Entering event state, Internal fault event
      OB80_FLT_ID : Byte;   // 16#XX, Fault identifcation code
      OB80_PRIORITY : Byte;   // Priority of OB Execution
      OB80_OB_NUMBR : Byte;   // 80 (Organization block 80, OB80)
      OB80_RESERVED_1 : Byte;   // Reserved for system
      OB80_RESERVED_2 : Byte;   // Reserved for system
      OB80_ERROR_INFO : Word;   // Error information on event
      OB80_ERR_EV_CLASS : Byte;   // Class of event causing error
      OB80_ERR_EV_NUM : Byte;   // Number of event causing error
      OB80_OB_PRIORITY : Byte;   // Priority of OB causing error
      OB80_OB_NUM : Byte;   // Number of OB causing error
      OB80_DATE_TIME : Date_And_Time;   // Date and time OB80 started
   END_VAR
BEGIN
END_ORGANIZATION_BLOCK

ORGANIZATION_BLOCK "RACK_FLT"   // OB86, LAD
TITLE = "Loss Of Rack Fault"
{ S7_Optimized_Access := 'FALSE' }
VERSION : 0.1
   VAR_TEMP
      OB86_EV_CLASS : Byte;   // 16#38/39 Event class 3
      OB86_FLT_ID : Byte;   // 16#C1/C4/C5, Fault identification code
      OB86_PRIORITY : Byte;   // Priority of OB Execution
      OB86_OB_NUMBR : Byte;   // 86 (Organization block 86, OB86)
      OB86_RESERVED_1 : Byte;   // Reserved for system
      OB86_RESERVED_2 : Byte;   // Reserved for system
      OB86_MDL_ADDR : Word;   // Base address of IM module in rack with fault
      OB86_RACKS_FLTD : Array[0..31] of Bool;   // Racks in fault
      OB86_DATE_TIME : Date_And_Time;   // Date and time OB86 started
   END_VAR
BEGIN
END_ORGANIZATION_BLOCK

ORGANIZATION_BLOCK "COMM_FLT"   // OB87, LAD
TITLE = "Communication Fault"
{ S7_Optimized_Access := 'FALSE' }
VERSION : 0.1
   VAR_TEMP
      OB87_EV_CLASS : Byte;   // 16#39 Event class 3
      OB87_FLT_ID : Byte;   // 16#XX, Fault identifcation code
      OB87_PRIORITY : Byte;   // Priority of OB Execution
      OB87_OB_NUMBR : Byte;   // 87 (Organization block 87, OB87)
      OB87_RESERVED_1 : Byte;   // Reserved for system
      OB87_RESERVED_2 : Byte;   // Reserved for system
      OB87_RESERVED_3 : Word;   // Reserved for system
      OB87_RESERVED_4 : DWord;   // Reserved for system
      OB87_DATE_TIME : Date_And_Time;   // Date and time OB87 started
   END_VAR
BEGIN
END_ORGANIZATION_BLOCK

ORGANIZATION_BLOCK "PROG_ERR"   // OB121, LAD
TITLE = "Programming Error"
{ S7_Optimized_Access := 'FALSE' }
VERSION : 0.1
   VAR_TEMP
      OB121_EV_CLASS : Byte;   // 16#25, Event class 2, Entering event state, Internal fault event
      OB121_SW_FLT : Byte;   // 16#XX Software programming fault
      OB121_PRIORITY : Byte;   // Priority of OB Execution
      OB121_OB_NUMBR : Byte;   // 121 (Organization block 121, OB121)
      OB121_BLK_TYPE : Byte;   // 16#88/8A/8B/8C/8E Type of block fault occured in
      OB121_RESERVED_1 : Byte;   // Reserved for system
      OB121_FLT_REG : Word;   // 16#XX Specific register that caused fault
      OB121_BLK_NUM : Word;   // Number of block that programming fault occured in
      OB121_PRG_ADDR : Word;   // Address in block where programming fault occured
      OB121_DATE_TIME : Date_And_Time;   // Date and time OB121 started
   END_VAR
BEGIN
END_ORGANIZATION_BLOCK

ORGANIZATION_BLOCK "MOD_ERR"   // OB122, LAD
TITLE = "Module Access Error"
{ S7_Optimized_Access := 'FALSE' }
VERSION : 0.1
   VAR_TEMP
      OB122_EV_CLASS : Byte;   // 16#29, Event class 2, Entering event state, Internal fault event
      OB122_SW_FLT : Byte;   // 16#XX Software error code
      OB122_PRIORITY : Byte;   // Priority of OB Execution
      OB122_OB_NUMBR : Byte;   // 122 (Organization block 122, OB122)
      OB122_BLK_TYPE : Byte;   // 16#88/8C/8E Type of block fault occured in
      OB122_MEM_AREA : Byte;   // Memory area where access error occured
      OB122_MEM_ADDR : Word;   // Memory address where access error occured
      OB122_BLK_NUM : Word;   // Block number in which error occured
      OB122_PRG_ADDR : Word;   // Program address where error occured
      OB122_DATE_TIME : Date_And_Time;   // Date and time OB1 started
   END_VAR
BEGIN
END_ORGANIZATION_BLOCK

// folder: Calculation

FUNCTION_BLOCK "FB_CalculateFlow"   // FB4, SCL
{ S7_Optimized_Access := 'FALSE' }
VERSION : 0.1
   VAR_INPUT
      PumpSpeed : Real;   // Speed [%]
   END_VAR
   VAR_OUTPUT
      Flow : Real;   // Flow [m3/h]
   END_VAR
BEGIN
   //
   // In this case, I am using an 8 inch diameter pipe which has a maximum flow of 454.2 m3 / h.
   // If we do simple calculate 100% - 454.2m3/h, so 1% is 4.542 m3/h.
   // 
   #Flow := #PumpSpeed * 4.542;
END_FUNCTION_BLOCK

FUNCTION_BLOCK "FB_FillingTankT1"   // FB5, SCL
{ S7_Optimized_Access := 'FALSE' }
VERSION : 0.1
   VAR_INPUT
      UV_1 : Bool;   // 0 - Valve close, 1 - Valve open
      FI_1 : Real;   // Measured Flow [m3/h]
      TRIGGER : Bool;   // 1hz
   END_VAR
   VAR_OUTPUT
      LI_1 : Real;   // Calculate level of fluid in tank 1
   END_VAR
   VAR
      SignalOld : Bool;
      CalcFI_1 : Real;
   END_VAR
   VAR_TEMP
      Edge : Bool;
   END_VAR
BEGIN
   // Positive edge detection
   #Edge := #TRIGGER AND NOT #SignalOld;
   #SignalOld := #TRIGGER;
   #CalcFI_1 := (#FI_1 * 1000.0) / 3600.0;

   IF (#UV_1) THEN
       IF (#Edge) THEN
           #LI_1 := #LI_1 + (189.25 - #CalcFI_1);
       END_IF;
   ELSIF (#UV_1 = FALSE) THEN
       IF (#Edge) THEN
           #LI_1 := #LI_1 - #CalcFI_1;
       END_IF;
   END_IF;
END_FUNCTION_BLOCK

FUNCTION_BLOCK "FB_FillingTankT2"   // FB6, SCL
{ S7_Optimized_Access := 'FALSE' }
VERSION : 0.1
   VAR_INPUT
      FI_1 : Real;   // Measured Flow [m3/h]
      FI_2 : Real;   // Measured Flow [m3/h]
      P3_Run : Bool;   // Dosing chemicals
      TRIGGER : Bool;   // 1hz
   END_VAR
   VAR_OUTPUT
      LI_2 : Real;   // Calculate level of fluid in tank 2
   END_VAR
   VAR
      SignalOld : Bool;
      CalcFI_1 : Real;
      CalcFI_2 : Real;
   END_VAR
   VAR_TEMP
      Edge : Bool;
   END_VAR
   VAR CONSTANT
      Chemicals : Real := 17.03;   // Amount of chemocal fluid added every second [l]
   END_VAR
BEGIN
   // Positive edge detection
   #Edge := #TRIGGER AND NOT #SignalOld;
   #SignalOld := #TRIGGER;
   #CalcFI_1 := (#FI_1 * 1000.0) / 3600.0;
   #CalcFI_2 := (#FI_2 * 1000.0) / 3600.0;

   IF (#Edge) THEN
       #LI_2 := #LI_2 + #CalcFI_1;
       #LI_2 := #LI_2 - #CalcFI_2;
       IF (#P3_Run) THEN
           #LI_2 := #LI_2 + #Chemicals;
       END_IF;
   END_IF;
END_FUNCTION_BLOCK

FUNCTION_BLOCK "FB_PhCalculation"   // FB8, SCL
{ S7_Optimized_Access := 'FALSE' }
VERSION : 0.1
   VAR_INPUT
      PhInputVal : Real;   // Input Random Ph Value
      P3_Run : Bool;   // Running signal from pump P3
      AI_1_SP : Real;   // Setpoint falue of Ph in Tank 3
      TRIGGER : Bool;   // 1Hz
   END_VAR
   VAR_OUTPUT
      AI_1 : Real;   // Calculated Ph in Tank 3
      ErrorValue : Bool;   // Value out of range (0-10) [Ph]
   END_VAR
   VAR
      SignalOld : Bool;
   END_VAR
   VAR_TEMP
      Edge : Bool;
      FirstScan : Bool;
   END_VAR
BEGIN
   // Positive edge detection
   #Edge := #TRIGGER AND NOT #SignalOld;
   #SignalOld := #TRIGGER;

   IF (#P3_Run AND #FirstScan = FALSE) THEN
       #FirstScan := TRUE;
       #AI_1 := #PhInputVal + 0.2;
   END_IF;

   IF (#Edge AND #P3_Run AND #FirstScan) THEN
       IF (#AI_1 < #AI_1_SP) THEN
           #AI_1 := #AI_1 + 0.2;
       ELSIF (#AI_1 > #AI_1_SP) THEN
           #AI_1 := #AI_1_SP;
       END_IF;
   END_IF;

   IF (#P3_Run = FALSE) THEN
       #FirstScan := FALSE;
   END_IF;
END_FUNCTION_BLOCK

FUNCTION_BLOCK "FB_EmptyingCT"   // FB9, SCL
{ S7_Optimized_Access := 'FALSE' }
VERSION : 0.1
   VAR_INPUT
      StartFilling : Bool;   // Start signal
      CTCapacity : Real;   // Chemical Tank Capacity [m3]
      FillTank : Bool;   // Fill Chemical Tank
      LowLevel : Bool;
      TRIGGER : Bool;
   END_VAR
   VAR_OUTPUT
      TankEmpty : Bool;   // Chemical Tank is Empty
      CalcCapacity : Real;
   END_VAR
   VAR
      SignalOld : Bool;
   END_VAR
   VAR_TEMP
      Edge : Bool;
   END_VAR
   VAR CONSTANT
      ChemicalsDose : Real := 17.03;   // Chemicals dose in every second
   END_VAR
BEGIN
   // Positive edge detection
   #Edge := #TRIGGER AND NOT #SignalOld;
   #SignalOld := #TRIGGER;


   IF (#FillTank) THEN
       #TankEmpty := FALSE;
       #CalcCapacity := #CTCapacity;
   END_IF;

   IF (#LowLevel) THEN
       #TankEmpty := TRUE;

   ELSIF(#LowLevel = FALSE)THEN
       IF (#StartFilling AND #Edge) THEN
           #CalcCapacity := #CTCapacity - #ChemicalsDose;
       END_IF;

   END_IF;
END_FUNCTION_BLOCK

// folder: Measuring Points

FUNCTION "Analogs" : Void   // FC4, LAD
{ S7_Optimized_Access := 'FALSE' }
VERSION : 0.1
BEGIN

REGION Network 1: LI_1 - Tank 1 Level
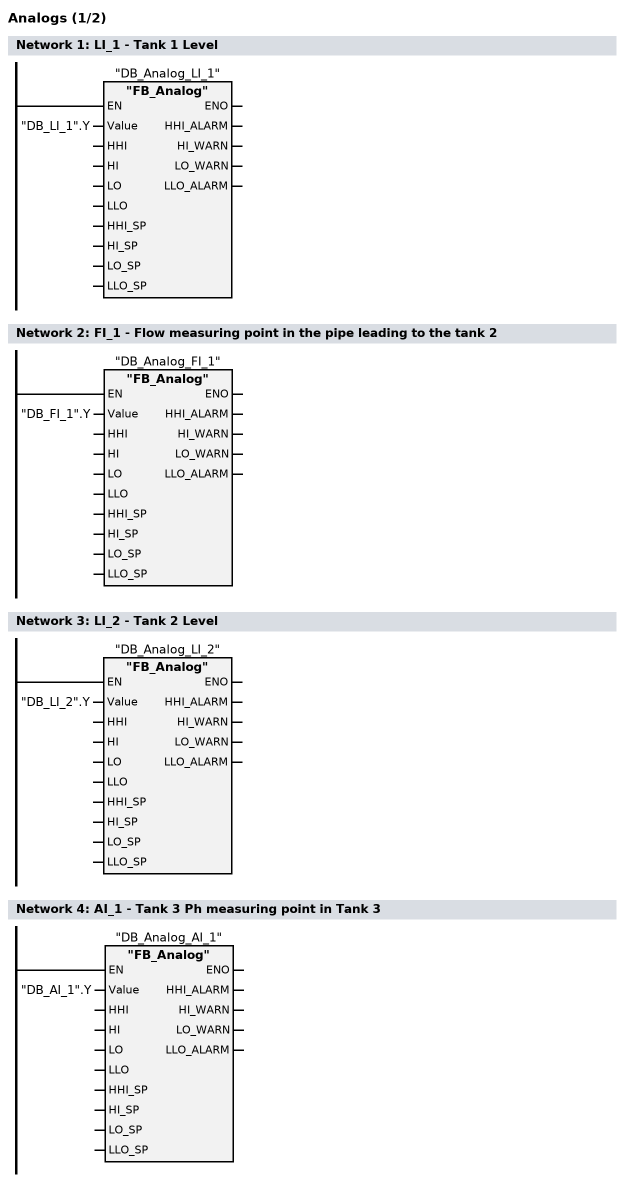
   RUNG wire#powerrail
      "DB_Analog_LI_1"(Value := "DB_LI_1".Y, HHI :=, HI :=, LO :=, LLO :=, HHI_SP :=, HI_SP :=, LO_SP :=, LLO_SP :=, HHI_ALARM =>, HI_WARN =>, LO_WARN =>, LLO_ALARM =>)
   END_RUNG
   // the same network as SCL:
   "DB_Analog_LI_1"(Value := "DB_LI_1".Y);   // "FB_Analog"
END_REGION

REGION Network 2: FI_1 - Flow measuring point in the pipe leading to the tank 2
   RUNG wire#powerrail
      "DB_Analog_FI_1"(Value := "DB_FI_1".Y, HHI :=, HI :=, LO :=, LLO :=, HHI_SP :=, HI_SP :=, LO_SP :=, LLO_SP :=, HHI_ALARM =>, HI_WARN =>, LO_WARN =>, LLO_ALARM =>)
   END_RUNG
   // the same network as SCL:
   "DB_Analog_FI_1"(Value := "DB_FI_1".Y);   // "FB_Analog"
END_REGION

REGION Network 3: LI_2 - Tank 2 Level
   RUNG wire#powerrail
      "DB_Analog_LI_2"(Value := "DB_LI_2".Y, HHI :=, HI :=, LO :=, LLO :=, HHI_SP :=, HI_SP :=, LO_SP :=, LLO_SP :=, HHI_ALARM =>, HI_WARN =>, LO_WARN =>, LLO_ALARM =>)
   END_RUNG
   // the same network as SCL:
   "DB_Analog_LI_2"(Value := "DB_LI_2".Y);   // "FB_Analog"
END_REGION

REGION Network 4: AI_1 - Tank 3 Ph measuring point in Tank 3
   RUNG wire#powerrail
      "DB_Analog_AI_1"(Value := "DB_AI_1".Y, HHI :=, HI :=, LO :=, LLO :=, HHI_SP :=, HI_SP :=, LO_SP :=, LLO_SP :=, HHI_ALARM =>, HI_WARN =>, LO_WARN =>, LLO_ALARM =>)
   END_RUNG
   // the same network as SCL:
   "DB_Analog_AI_1"(Value := "DB_AI_1".Y);   // "FB_Analog"
END_REGION

REGION Network 5: FI_2 - Flow measuring point at the end of the line
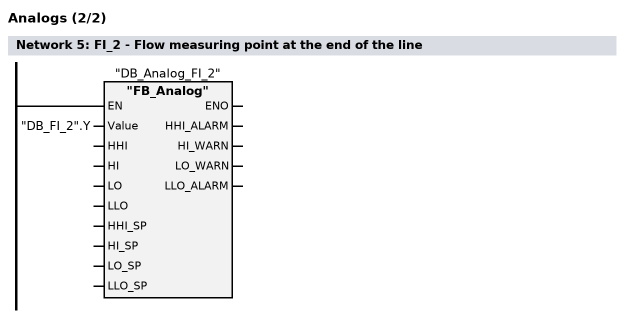
   RUNG wire#powerrail
      "DB_Analog_FI_2"(Value := "DB_FI_2".Y, HHI :=, HI :=, LO :=, LLO :=, HHI_SP :=, HI_SP :=, LO_SP :=, LLO_SP :=, HHI_ALARM =>, HI_WARN =>, LO_WARN =>, LLO_ALARM =>)
   END_RUNG
   // the same network as SCL:
   "DB_Analog_FI_2"(Value := "DB_FI_2".Y);   // "FB_Analog"
END_REGION
END_FUNCTION

FUNCTION "Measuring Transducers" : Void   // FC7, FBD
{ S7_Optimized_Access := 'FALSE' }
VERSION : 0.1
BEGIN

REGION Network 1: LI_1 - Tank 1 Level
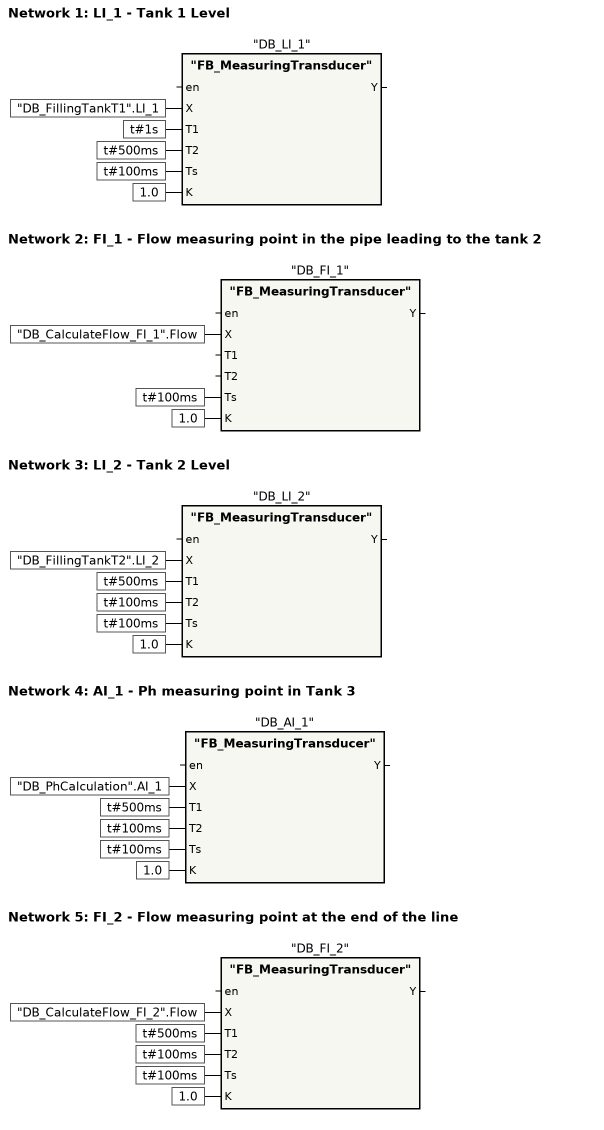
   "DB_LI_1"(X := "DB_FillingTankT1".LI_1, T1 := t#1s, T2 := t#500ms, Ts := t#100ms, K := 1.0);   // "FB_MeasuringTransducer"
END_REGION

REGION Network 2: FI_1 - Flow measuring point in the pipe leading to the tank 2
   "DB_FI_1"(X := "DB_CalculateFlow_FI_1".Flow, Ts := t#100ms, K := 1.0);   // "FB_MeasuringTransducer"
END_REGION

REGION Network 3: LI_2 - Tank 2 Level
   "DB_LI_2"(X := "DB_FillingTankT2".LI_2, T1 := t#500ms, T2 := t#100ms, Ts := t#100ms, K := 1.0);   // "FB_MeasuringTransducer"
END_REGION

REGION Network 4: AI_1 - Ph measuring point in Tank 3
   "DB_AI_1"(X := "DB_PhCalculation".AI_1, T1 := t#500ms, T2 := t#100ms, Ts := t#100ms, K := 1.0);   // "FB_MeasuringTransducer"
END_REGION

REGION Network 5: FI_2 - Flow measuring point at the end of the line
   "DB_FI_2"(X := "DB_CalculateFlow_FI_2".Flow, T1 := t#500ms, T2 := t#100ms, Ts := t#100ms, K := 1.0);   // "FB_MeasuringTransducer"
END_REGION
END_FUNCTION

// folder: Program files

FUNCTION "FC_FILL_T1" : Void   // FC2, LAD
TITLE = Filling tank T1
{ S7_Optimized_Access := 'FALSE' }
VERSION : 0.1
BEGIN

REGION Network 1: Start filling proces
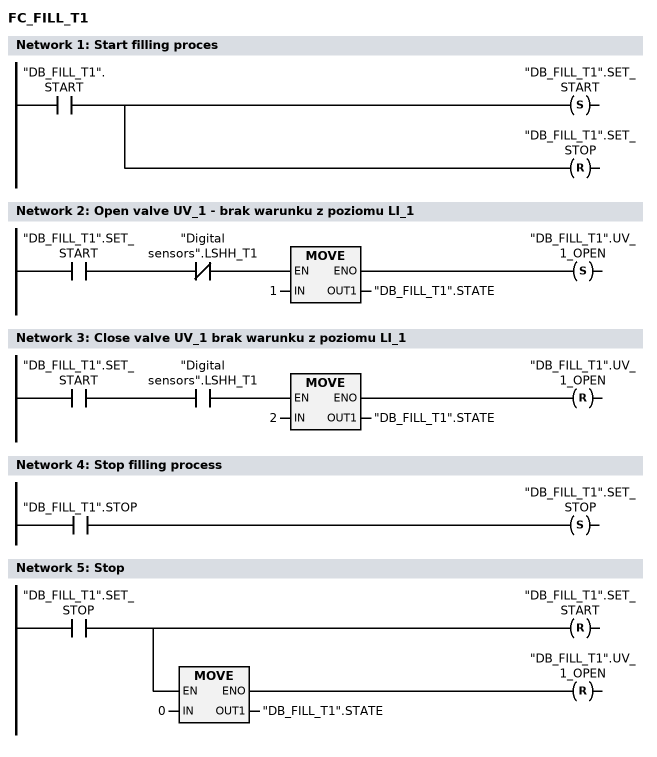
   RUNG wire#powerrail
      Contact( "DB_FILL_T1".START )
      wire#w1
      S_Coil( "DB_FILL_T1".SET_START )
   END_RUNG
   RUNG wire#w1
      R_Coil( "DB_FILL_T1".SET_STOP )
   END_RUNG
   // the same network as SCL:
   IF "DB_FILL_T1".START THEN
       "DB_FILL_T1".SET_START := TRUE;
       "DB_FILL_T1".SET_STOP := FALSE;
   END_IF;
END_REGION

REGION Network 2: Open valve UV_1 - brak warunku z poziomu LI_1
   RUNG wire#powerrail
      Contact( "DB_FILL_T1".SET_START )
      I_Contact( "Digital sensors".LSHH_T1 )
      { S7_GenerateENO := "TRUE" } Move(in := 1, out1 => "DB_FILL_T1".STATE)
      S_Coil( "DB_FILL_T1".UV_1_OPEN )
   END_RUNG
   // the same network as SCL:
   // ENO of a box is taken as its EN; it also drops when the box reports an error
   IF "DB_FILL_T1".SET_START AND NOT "Digital sensors".LSHH_T1 THEN
       "DB_FILL_T1".STATE := 1;
       "DB_FILL_T1".UV_1_OPEN := TRUE;
   END_IF;
END_REGION

REGION Network 3: Close valve UV_1 brak warunku z poziomu LI_1
   RUNG wire#powerrail
      Contact( "DB_FILL_T1".SET_START )
      Contact( "Digital sensors".LSHH_T1 )
      { S7_GenerateENO := "TRUE" } Move(in := 2, out1 => "DB_FILL_T1".STATE)
      R_Coil( "DB_FILL_T1".UV_1_OPEN )
   END_RUNG
   // the same network as SCL:
   // ENO of a box is taken as its EN; it also drops when the box reports an error
   IF "DB_FILL_T1".SET_START AND "Digital sensors".LSHH_T1 THEN
       "DB_FILL_T1".STATE := 2;
       "DB_FILL_T1".UV_1_OPEN := FALSE;
   END_IF;
END_REGION

REGION Network 4: Stop filling process
   RUNG wire#powerrail
      Contact( "DB_FILL_T1".STOP )
      S_Coil( "DB_FILL_T1".SET_STOP )
   END_RUNG
   // the same network as SCL:
   IF "DB_FILL_T1".STOP THEN "DB_FILL_T1".SET_STOP := TRUE; END_IF;
END_REGION

REGION Network 5: Stop
   RUNG wire#powerrail
      Contact( "DB_FILL_T1".SET_STOP )
      wire#w1
      R_Coil( "DB_FILL_T1".SET_START )
   END_RUNG
   RUNG wire#w1
      { S7_GenerateENO := "TRUE" } Move(in := 0, out1 => "DB_FILL_T1".STATE)
      R_Coil( "DB_FILL_T1".UV_1_OPEN )
   END_RUNG
   // the same network as SCL:
   // ENO of a box is taken as its EN; it also drops when the box reports an error
   IF "DB_FILL_T1".SET_STOP THEN
       "DB_FILL_T1".SET_START := FALSE;
       "DB_FILL_T1".STATE := 0;
       "DB_FILL_T1".UV_1_OPEN := FALSE;
   END_IF;
END_REGION
END_FUNCTION

FUNCTION "FC_TRANSFER_TO_T2" : Void   // FC3, LAD
TITLE = Transfer to Tank T2
{ S7_Optimized_Access := 'FALSE' }
VERSION : 0.1
   VAR_TEMP
      PhVal : Bool;
   END_VAR
   VAR_TEMP   // added for the SCL form of the ladder/FBD networks
      _w1 : Bool;
      _w2 : Bool;
   END_VAR
BEGIN

REGION Network 1: Start signal from SCADA
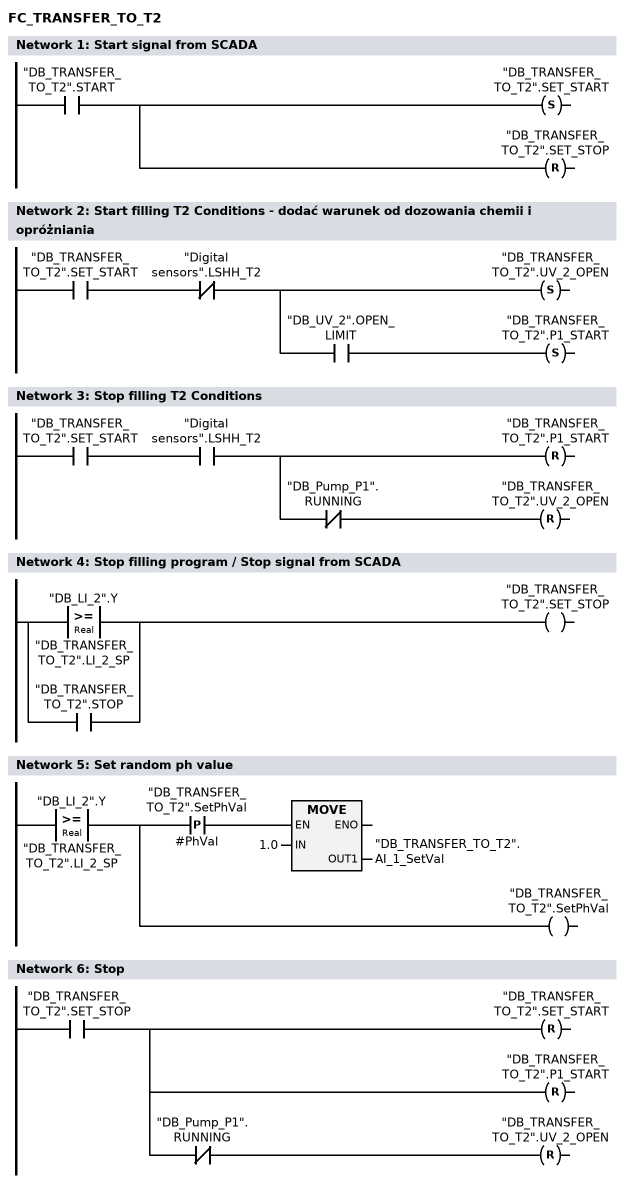
   RUNG wire#powerrail
      Contact( "DB_TRANSFER_TO_T2".START )
      wire#w1
      S_Coil( "DB_TRANSFER_TO_T2".SET_START )
   END_RUNG
   RUNG wire#w1
      R_Coil( "DB_TRANSFER_TO_T2".SET_STOP )
   END_RUNG
   // the same network as SCL:
   IF "DB_TRANSFER_TO_T2".START THEN
       "DB_TRANSFER_TO_T2".SET_START := TRUE;
       "DB_TRANSFER_TO_T2".SET_STOP := FALSE;
   END_IF;
END_REGION

REGION Network 2: Start filling T2 Conditions - dodać warunek od dozowania chemii i opróżniania
   RUNG wire#powerrail
      Contact( "DB_TRANSFER_TO_T2".SET_START )
      I_Contact( "Digital sensors".LSHH_T2 )
      wire#w1
      S_Coil( "DB_TRANSFER_TO_T2".UV_2_OPEN )
   END_RUNG
   RUNG wire#w1
      Contact( "DB_UV_2".OPEN_LIMIT )
      S_Coil( "DB_TRANSFER_TO_T2".P1_START )
   END_RUNG
   // the same network as SCL:
   #_w1 := "DB_TRANSFER_TO_T2".SET_START AND NOT "Digital sensors".LSHH_T2;
   IF #_w1 THEN "DB_TRANSFER_TO_T2".UV_2_OPEN := TRUE; END_IF;
   IF #_w1 AND "DB_UV_2".OPEN_LIMIT THEN "DB_TRANSFER_TO_T2".P1_START := TRUE; END_IF;
END_REGION

REGION Network 3: Stop filling T2 Conditions
   RUNG wire#powerrail
      Contact( "DB_TRANSFER_TO_T2".SET_START )
      Contact( "Digital sensors".LSHH_T2 )
      wire#w1
      R_Coil( "DB_TRANSFER_TO_T2".P1_START )
   END_RUNG
   RUNG wire#w1
      I_Contact( "DB_Pump_P1".RUNNING )
      R_Coil( "DB_TRANSFER_TO_T2".UV_2_OPEN )
   END_RUNG
   // the same network as SCL:
   #_w1 := "DB_TRANSFER_TO_T2".SET_START AND "Digital sensors".LSHH_T2;
   IF #_w1 THEN "DB_TRANSFER_TO_T2".P1_START := FALSE; END_IF;
   IF #_w1 AND NOT "DB_Pump_P1".RUNNING THEN "DB_TRANSFER_TO_T2".UV_2_OPEN := FALSE; END_IF;
END_REGION

REGION Network 4: Stop filling program / Stop signal from SCADA
   RUNG wire#powerrail
      { S7_Templates := "SrcType := Real" } GE_Contact(in1 := "DB_LI_2".Y, in2 := "DB_TRANSFER_TO_T2".LI_2_SP)
      wire#w1
      Coil( "DB_TRANSFER_TO_T2".SET_STOP )
   END_RUNG
   RUNG wire#powerrail
      Contact( "DB_TRANSFER_TO_T2".STOP )
   END_RUNG wire#w1
   // the same network as SCL:
   "DB_TRANSFER_TO_T2".SET_STOP := ("DB_LI_2".Y >= "DB_TRANSFER_TO_T2".LI_2_SP) OR "DB_TRANSFER_TO_T2".STOP;
END_REGION

REGION Network 5: Set random ph value
   RUNG wire#powerrail
      { S7_Templates := "SrcType := Real" } GE_Contact(in1 := "DB_LI_2".Y, in2 := "DB_TRANSFER_TO_T2".LI_2_SP)
      wire#w1
      P_Contact(operand := "DB_TRANSFER_TO_T2".SetPhVal, bit := #PhVal)
      { S7_GenerateENO := "TRUE" } Move(in := 1.0, out1 => "DB_TRANSFER_TO_T2".AI_1_SetVal)
   END_RUNG
   RUNG wire#w1
      Coil( "DB_TRANSFER_TO_T2".SetPhVal )
   END_RUNG
   // the same network as SCL:
   #_w1 := "DB_LI_2".Y >= "DB_TRANSFER_TO_T2".LI_2_SP;
   #_w2 := #_w1 AND "DB_TRANSFER_TO_T2".SetPhVal AND NOT #PhVal;   // rising edge of "DB_TRANSFER_TO_T2".SetPhVal
   #PhVal := "DB_TRANSFER_TO_T2".SetPhVal;
   IF #_w2 THEN "DB_TRANSFER_TO_T2".AI_1_SetVal := 1.0; END_IF;
   "DB_TRANSFER_TO_T2".SetPhVal := #_w1;
END_REGION

REGION Network 6: Stop
   RUNG wire#powerrail
      Contact( "DB_TRANSFER_TO_T2".SET_STOP )
      wire#w1
      R_Coil( "DB_TRANSFER_TO_T2".SET_START )
   END_RUNG
   RUNG wire#w1
      R_Coil( "DB_TRANSFER_TO_T2".P1_START )
   END_RUNG
   RUNG wire#w1
      I_Contact( "DB_Pump_P1".RUNNING )
      R_Coil( "DB_TRANSFER_TO_T2".UV_2_OPEN )
   END_RUNG
   // the same network as SCL:
   IF "DB_TRANSFER_TO_T2".SET_STOP THEN
       "DB_TRANSFER_TO_T2".SET_START := FALSE;
       "DB_TRANSFER_TO_T2".P1_START := FALSE;
   END_IF;
   IF "DB_TRANSFER_TO_T2".SET_STOP AND NOT "DB_Pump_P1".RUNNING THEN
       "DB_TRANSFER_TO_T2".UV_2_OPEN := FALSE;
   END_IF;
END_REGION
END_FUNCTION

FUNCTION "FC_DOSE_CHEMICALS" : Void   // FC5, LAD
TITLE = Dosing Chemicals to Tank 2
{ S7_Optimized_Access := 'FALSE' }
VERSION : 0.1
   VAR_TEMP   // added for the SCL form of the ladder/FBD networks
      _w1 : Bool;
   END_VAR
BEGIN

REGION Network 1: Start
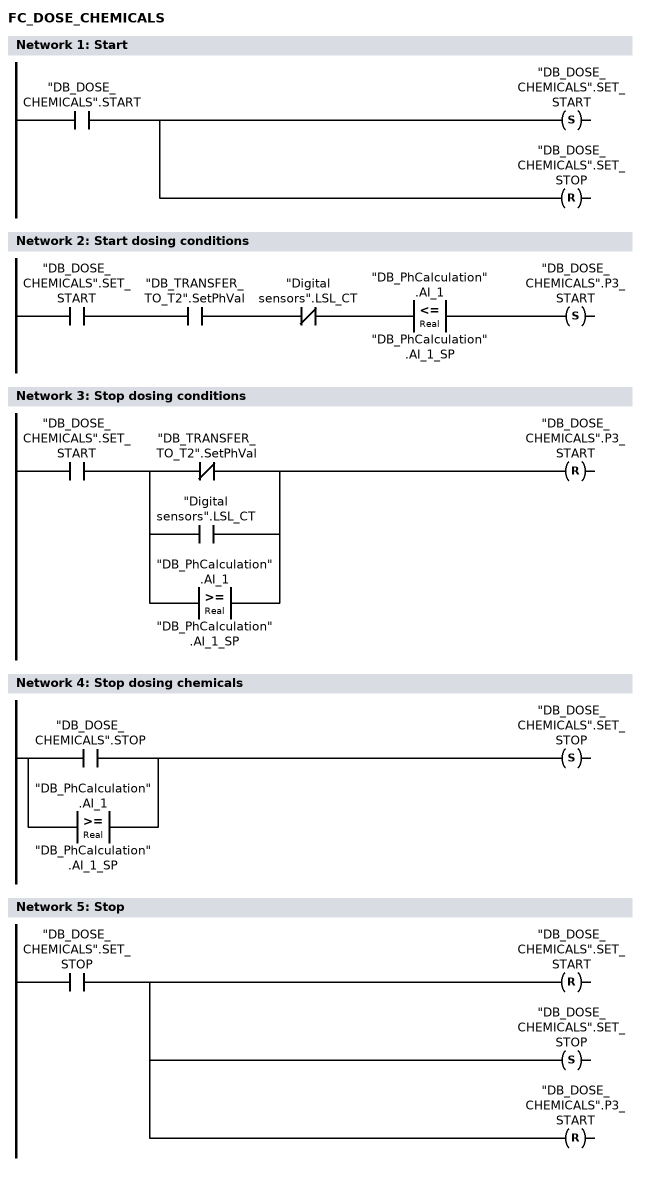
   RUNG wire#powerrail
      Contact( "DB_DOSE_CHEMICALS".START )
      wire#w1
      S_Coil( "DB_DOSE_CHEMICALS".SET_START )
   END_RUNG
   RUNG wire#w1
      R_Coil( "DB_DOSE_CHEMICALS".SET_STOP )
   END_RUNG
   // the same network as SCL:
   IF "DB_DOSE_CHEMICALS".START THEN
       "DB_DOSE_CHEMICALS".SET_START := TRUE;
       "DB_DOSE_CHEMICALS".SET_STOP := FALSE;
   END_IF;
END_REGION

REGION Network 2: Start dosing conditions
   RUNG wire#powerrail
      Contact( "DB_DOSE_CHEMICALS".SET_START )
      Contact( "DB_TRANSFER_TO_T2".SetPhVal )
      I_Contact( "Digital sensors".LSL_CT )
      { S7_Templates := "SrcType := Real" } LE_Contact(in1 := "DB_PhCalculation".AI_1, in2 := "DB_PhCalculation".AI_1_SP)
      S_Coil( "DB_DOSE_CHEMICALS".P3_START )
   END_RUNG
   // the same network as SCL:
   IF "DB_DOSE_CHEMICALS".SET_START AND "DB_TRANSFER_TO_T2".SetPhVal AND NOT "Digital sensors".LSL_CT AND ("DB_PhCalculation".AI_1 <= "DB_PhCalculation".AI_1_SP) THEN
       "DB_DOSE_CHEMICALS".P3_START := TRUE;
   END_IF;
END_REGION

REGION Network 3: Stop dosing conditions
   RUNG wire#powerrail
      Contact( "DB_DOSE_CHEMICALS".SET_START )
      wire#w1
      I_Contact( "DB_TRANSFER_TO_T2".SetPhVal )
      wire#w2
      R_Coil( "DB_DOSE_CHEMICALS".P3_START )
   END_RUNG
   RUNG wire#w1
      Contact( "Digital sensors".LSL_CT )
   END_RUNG wire#w2
   RUNG wire#w1
      { S7_Templates := "SrcType := Real" } GE_Contact(in1 := "DB_PhCalculation".AI_1, in2 := "DB_PhCalculation".AI_1_SP)
   END_RUNG wire#w2
   // the same network as SCL:
   IF "DB_DOSE_CHEMICALS".SET_START AND (NOT "DB_TRANSFER_TO_T2".SetPhVal OR "Digital sensors".LSL_CT OR ("DB_PhCalculation".AI_1 >= "DB_PhCalculation".AI_1_SP)) THEN
       "DB_DOSE_CHEMICALS".P3_START := FALSE;
   END_IF;
END_REGION

REGION Network 4: Stop dosing chemicals
   RUNG wire#powerrail
      Contact( "DB_DOSE_CHEMICALS".STOP )
      wire#w1
      S_Coil( "DB_DOSE_CHEMICALS".SET_STOP )
   END_RUNG
   RUNG wire#powerrail
      { S7_Templates := "SrcType := Real" } GE_Contact(in1 := "DB_PhCalculation".AI_1, in2 := "DB_PhCalculation".AI_1_SP)
   END_RUNG wire#w1
   // the same network as SCL:
   IF "DB_DOSE_CHEMICALS".STOP OR ("DB_PhCalculation".AI_1 >= "DB_PhCalculation".AI_1_SP) THEN
       "DB_DOSE_CHEMICALS".SET_STOP := TRUE;
   END_IF;
END_REGION

REGION Network 5: Stop
   RUNG wire#powerrail
      Contact( "DB_DOSE_CHEMICALS".SET_STOP )
      wire#w1
      R_Coil( "DB_DOSE_CHEMICALS".SET_START )
   END_RUNG
   RUNG wire#w1
      S_Coil( "DB_DOSE_CHEMICALS".SET_STOP )
   END_RUNG
   RUNG wire#w1
      R_Coil( "DB_DOSE_CHEMICALS".P3_START )
   END_RUNG
   // the same network as SCL:
   IF "DB_DOSE_CHEMICALS".SET_STOP THEN "DB_DOSE_CHEMICALS".SET_START := FALSE; END_IF;
   #_w1 := "DB_DOSE_CHEMICALS".SET_STOP;
   IF #_w1 THEN
       "DB_DOSE_CHEMICALS".SET_STOP := TRUE;
       "DB_DOSE_CHEMICALS".P3_START := FALSE;
   END_IF;
END_REGION
END_FUNCTION

FUNCTION "FC_EMPTYING_T2" : Void   // FC6, LAD
TITLE = Emptyking Tank T2 - Finish process
{ S7_Optimized_Access := 'FALSE' }
VERSION : 0.1
BEGIN

REGION Network 1: Set start signal
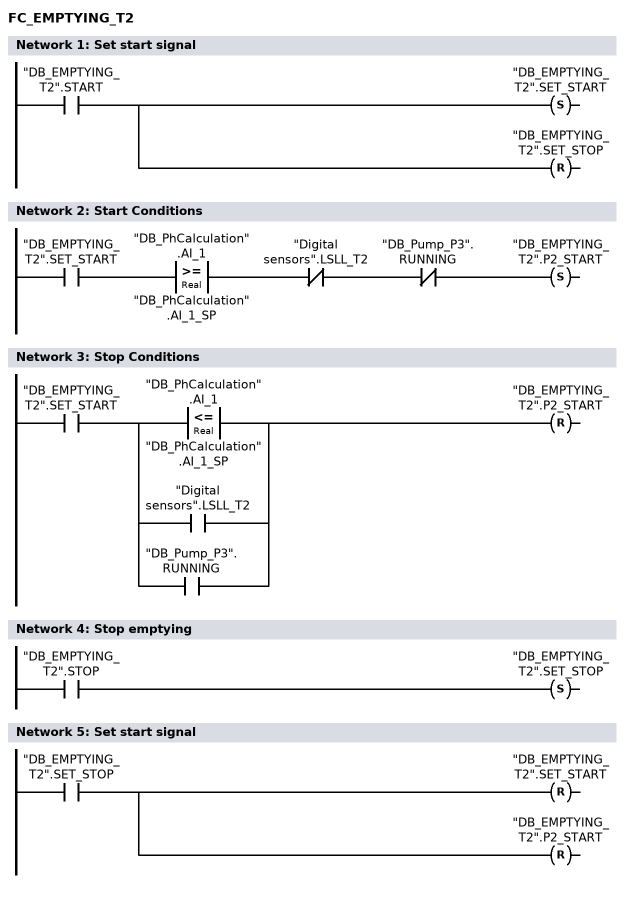
   RUNG wire#powerrail
      Contact( "DB_EMPTYING_T2".START )
      wire#w1
      S_Coil( "DB_EMPTYING_T2".SET_START )
   END_RUNG
   RUNG wire#w1
      R_Coil( "DB_EMPTYING_T2".SET_STOP )
   END_RUNG
   // the same network as SCL:
   IF "DB_EMPTYING_T2".START THEN
       "DB_EMPTYING_T2".SET_START := TRUE;
       "DB_EMPTYING_T2".SET_STOP := FALSE;
   END_IF;
END_REGION

REGION Network 2: Start Conditions
   RUNG wire#powerrail
      Contact( "DB_EMPTYING_T2".SET_START )
      { S7_Templates := "SrcType := Real" } GE_Contact(in1 := "DB_PhCalculation".AI_1, in2 := "DB_PhCalculation".AI_1_SP)
      I_Contact( "Digital sensors".LSLL_T2 )
      I_Contact( "DB_Pump_P3".RUNNING )
      S_Coil( "DB_EMPTYING_T2".P2_START )
   END_RUNG
   // the same network as SCL:
   IF "DB_EMPTYING_T2".SET_START AND ("DB_PhCalculation".AI_1 >= "DB_PhCalculation".AI_1_SP) AND NOT "Digital sensors".LSLL_T2 AND NOT "DB_Pump_P3".RUNNING THEN
       "DB_EMPTYING_T2".P2_START := TRUE;
   END_IF;
END_REGION

REGION Network 3: Stop Conditions
   RUNG wire#powerrail
      Contact( "DB_EMPTYING_T2".SET_START )
      wire#w1
      { S7_Templates := "SrcType := Real" } LE_Contact(in1 := "DB_PhCalculation".AI_1, in2 := "DB_PhCalculation".AI_1_SP)
      wire#w2
      R_Coil( "DB_EMPTYING_T2".P2_START )
   END_RUNG
   RUNG wire#w1
      Contact( "Digital sensors".LSLL_T2 )
   END_RUNG wire#w2
   RUNG wire#w1
      Contact( "DB_Pump_P3".RUNNING )
   END_RUNG wire#w2
   // the same network as SCL:
   IF "DB_EMPTYING_T2".SET_START AND (("DB_PhCalculation".AI_1 <= "DB_PhCalculation".AI_1_SP) OR "Digital sensors".LSLL_T2 OR "DB_Pump_P3".RUNNING) THEN
       "DB_EMPTYING_T2".P2_START := FALSE;
   END_IF;
END_REGION

REGION Network 4: Stop emptying
   RUNG wire#powerrail
      Contact( "DB_EMPTYING_T2".STOP )
      S_Coil( "DB_EMPTYING_T2".SET_STOP )
   END_RUNG
   // the same network as SCL:
   IF "DB_EMPTYING_T2".STOP THEN "DB_EMPTYING_T2".SET_STOP := TRUE; END_IF;
END_REGION

REGION Network 5: Set start signal
   RUNG wire#powerrail
      Contact( "DB_EMPTYING_T2".SET_STOP )
      wire#w1
      R_Coil( "DB_EMPTYING_T2".SET_START )
   END_RUNG
   RUNG wire#w1
      R_Coil( "DB_EMPTYING_T2".P2_START )
   END_RUNG
   // the same network as SCL:
   IF "DB_EMPTYING_T2".SET_STOP THEN
       "DB_EMPTYING_T2".SET_START := FALSE;
       "DB_EMPTYING_T2".P2_START := FALSE;
   END_IF;
END_REGION
END_FUNCTION

// ===== library types =====

// folder: LGF/4 Math operations

FUNCTION "LGF_RandomRange_Real" : Real   // FC10014, SCL
TITLE = LGF_RandomRange_Real
{ S7_Optimized_Access := 'TRUE' }
AUTHOR : Siemens_Digital_Industries
FAMILY : LGF
NAME : LGF_RandomRange_Real
// This function generates random numbers in defined limits (Datatype Real)
   VAR_INPUT
      minValue : Real;   // minimal Value random can reach / Minimum value of the range of the random number
      maxValue : Real;   // maximal Value random can reach / Maximum value of the range of the random number
   END_VAR
   VAR_OUTPUT
      error : Bool;   // Error if true
      status : Word;   // Status of the function
      subfunctionStatus : Word;   // Status or return value of called FB's, FCs and system blocks
   END_VAR
   VAR_TEMP
      tempTime : DTL;   // System time
      tempNanoSecondInDWord : DWord;   // UDINT converted to DWORD for access to individual bytes
      tempTimeStatus : Word;   // Status of the instruction RD_SYS_T
      tempRandomValue : DWord;   // Random-start-value
      tempNormReal : Real;   // normalized value
   END_VAR
   // Ret_Val : Returns random Real number in predefined range
   VAR CONSTANT
      ZERO : Real := 0.0;   // Zero value in case of error
      MAX_UDINT : UDInt := 4294967295;   // Maximum UDINT value
      SUB_STATUS_NO_ERROR : Word := 16#0000;   // Status: sub function call ends without error
      STATUS_FINISHED_NO_ERROR : Word := 16#0000;   // Status: Execution finished without errors
      ERR_MAX_LESS_MIN : Word := 16#8200;   // Error: The maximum limit number is smaller than the minimum limit number
      ERR_RD_SYS_T : Word := 16#8600;   // Error: System function Read system time returned an error
   END_VAR
BEGIN
   REGION Block info header
     //=============================================================================
     // SIEMENS AG / (c)Copyright 2017
     //-----------------------------------------------------------------------------
     // Title:            LGF_RandomRange_Real
     // Comment/Function: This function generates random numbers in defined limits (Datatype Real)
     // Library/Family:   LGF(Library General Functions)
     // Author:           Siemens Digital Industry Support
     // Tested with:      S7-PLCSIM Advanced V2.0 SP1
     // Engineering:      TIA Portal V15 Update 2
     // Restrictions:     ENO disabled - error handling done by error and status
     // Requirements:     PLC (S7-1200 / S7-1500)
     //-------------------------------------------------------------------------------
     // Change log table:
     // Version  | Date       | Expert in charge       | Changes applied
     //----------|------------|------------------------|------------------------------
     // 01.00.00 19.08.2015  Siemens Industry Online Support
     //                      First released version
     // 01.00.01 02.01.2017  Siemens Industry Online Support
     //                      Upgrade: TIA Portal V14 Update 1
     // 01.00.02 02.03.2017  Siemens Industry Online Support
     //                      Bugfix: FC number
     // 01.00.03 17.08.2018  Siemens Industry Online Support
     //                      Upgrade: TIA V15 Update 2
     // 01.00.04 23.11.2018  Siemens Industry Online Support
     //                      Upgrade: TIA V15.1
     // 01.01.00 13.11.2019  Siemens Industry Presales Support
     //                      Renamed from "LGF_RandomReal" to "LGF_RandomRange_Real"
     //                      Regions, commens and costants are added
     // 03.00.00 23.04.2020  Siemens Industry Support
     //                      Set version to V3.0.0, harmonize the version of the whole library
     //=============================================================================
   END_REGION

   REGION Validation
     // Check if the maximal Value is less than the minimal value
     IF (#minValue > #maxValue) THEN
       #error := true;
       #status := #ERR_MAX_LESS_MIN;
       #subfunctionStatus := #SUB_STATUS_NO_ERROR;
       #LGF_RandomRange_Real := #ZERO;
       RETURN;
     END_IF;

     // Read system time
     #tempTimeStatus := INT_TO_WORD(RD_SYS_T(#tempTime));

     // Check return variable for error
     IF (#tempTimeStatus <> #SUB_STATUS_NO_ERROR) THEN
       #error := true;
       #status := #ERR_RD_SYS_T;
       #subfunctionStatus := #tempTimeStatus;
       #LGF_RandomRange_Real := #ZERO;
       RETURN;
     END_IF;
   END_REGION

   REGION Calculating random number
     // Converting to double word so individual bytes can be addressed
     #tempNanoSecondInDWord := UDINT_TO_DWORD(#tempTime.NANOSECOND);

     // Calculate a random-start-value depending on the time
     #tempRandomValue.%B3 := #tempNanoSecondInDWord.%B0;
     #tempRandomValue.%B2 := #tempNanoSecondInDWord.%B1;
     #tempRandomValue.%B1 := #tempNanoSecondInDWord.%B2;
     #tempRandomValue.%B0 := #tempNanoSecondInDWord.%B3;

     // Norm the calculated random number: 0.0 <= #tempNormReal <= 1.0
     #tempNormReal := UDINT_TO_REAL(DWORD_TO_UDINT(#tempRandomValue)) / UDINT_TO_REAL(#MAX_UDINT);

     // Scale the tempNormReal to be in the range of maxValue and minValue
     #LGF_RandomRange_Real := ((#tempNormReal * (#maxValue - #minValue) + (#minValue)));

     #error := false;
     #status := #STATUS_FINISHED_NO_ERROR;
     #subfunctionStatus := #SUB_STATUS_NO_ERROR;
     // ENO mechanism is not used
     ENO := TRUE;
   END_REGION
END_FUNCTION

FUNCTION "LGF_RandomRange_UDInt" : UDInt   // FC10079, SCL
TITLE = LGF_RandomRange_UDInt
{ S7_Optimized_Access := 'TRUE' }
AUTHOR : Siemens_Digital_Industries
FAMILY : LGF
NAME : LGF_RandomRange_UDInt
// This function generates random numbers in defined limits (Datatype UDInt)
   VAR_INPUT
      minValue : UDInt;   // minimal Value random can reach / Minimum value of the range of the random number
      maxValue : UDInt;   // maximal Value random can reach / Maximum value of the range of the random number
   END_VAR
   VAR_OUTPUT
      error : Bool;   // Error if true
      status : Word;   // Status of the function
      subfunctionStatus : Word;   // Status or return value of called FB's, FCs and system blocks
   END_VAR
   VAR_TEMP
      tempTime : DTL;   // System time
      tempNanoSecondInDWord : DWord;   // UDINT converted to DWORD for access to individual bytes
      tempTimeStatus : Word;   // Status of the instruction RD_SYS_T
      tempRandomValue : DWord;   // Random-start-value
      tempNormReal : Real;   // Normalized value
   END_VAR
   // Ret_Val : Returns random UDInt number in a predefined range
   VAR CONSTANT
      ZERO : UDInt := 0;   // Zero value in case of error
      MAX_UDINT : UDInt := 4294967295 ;   // Maximum UDINT value
      SUB_STATUS_NO_ERROR : Word := 16#0000;   // Status: sub function call ends without error
      STATUS_FINISHED_NO_ERROR : Word := 16#0000;   // Status: Execution finished without errors
      ERR_MAX_LESS_MIN : Word := 16#8200;   // Error: The maximum limit number is smaller than the minimum limit number
      ERR_RD_SYS_T : Word := 16#8600;   // Error: System function Read system time returned an error
   END_VAR
BEGIN
   REGION Block info header
     //=============================================================================
     // SIEMENS AG / (c)Copyright 2019
     //-----------------------------------------------------------------------------
     // Title:            LGF_RandomRange_UDInt
     // Comment/Function: This function generates random numbers in defined limits (Datatype UDInt)
     // Library/Family:   LGF(Library General Functions)
     // Author:           Siemens Digital Industry Support
     // Tested with:      S7-PLCSIM Advanced V2.0 SP1
     // Engineering:      TIA Portal V15 Update 2
     // Restrictions:     ENO disabled - error handling done by error and status
     // Requirements:     PLC (S7-1200 / S7-1500)
     //-------------------------------------------------------------------------------
     // Change log table:
     // Version  | Date       | Expert in charge       | Changes applied
     //----------|------------|------------------------|------------------------------
     // 01.00.00 11.12.2019  Siemens Industry Online Support
     //                      First released version
     //                      copied from "LGF_RandomRange_DInt"
     // 03.00.00 23.04.2020  Siemens Industry Support
     //                      Set version to V3.0.0, harmonize the version of the whole library
     //=============================================================================
   END_REGION

   REGION Validation
     // Check if the maximal Value is less than the minimal value
     IF (#minValue > #maxValue) THEN
       #error := true;
       #status := #ERR_MAX_LESS_MIN;
       #subfunctionStatus := #SUB_STATUS_NO_ERROR;
       #LGF_RandomRange_UDInt := #ZERO;
       RETURN;
     END_IF;

     // Read system time
     #tempTimeStatus := INT_TO_WORD(RD_SYS_T(#tempTime));

     // Check return variable for error
     IF (#tempTimeStatus <> #SUB_STATUS_NO_ERROR) THEN
       #error := true;
       #status := #ERR_RD_SYS_T;
       #subfunctionStatus := #tempTimeStatus;
       #LGF_RandomRange_UDInt := #ZERO;
       RETURN;
     END_IF;
   END_REGION

   REGION Calculating random number
     // Converting to double word so individual bytes can be addressed
     #tempNanoSecondInDWord := UDINT_TO_DWORD(#tempTime.NANOSECOND);

     // Calculate a random-start-value depending on the time
     #tempRandomValue.%B3 := #tempNanoSecondInDWord.%B0;
     #tempRandomValue.%B2 := #tempNanoSecondInDWord.%B1;
     #tempRandomValue.%B1 := #tempNanoSecondInDWord.%B2;
     #tempRandomValue.%B0 := #tempNanoSecondInDWord.%B3;

     // Norm the calculated random number: 0.0 <= #tempNormReal <= 1.0
     #tempNormReal := UDINT_TO_REAL(DWORD_TO_UDINT(#tempRandomValue)) / UDINT_TO_REAL(#MAX_UDINT);

     // Scale the tempNormReal to be in the range of maxValue and minValue
     #LGF_RandomRange_UDInt := REAL_TO_UDINT((#tempNormReal * UDINT_TO_REAL(#maxValue - #minValue) + UDINT_TO_REAL(#minValue)));

     #error := false;
     #status := #STATUS_FINISHED_NO_ERROR;
     #subfunctionStatus := #SUB_STATUS_NO_ERROR;
     // ENO mechanism is not used
     ENO := TRUE;
   END_REGION
END_FUNCTION

FUNCTION "LGF_Random_DInt" : DInt   // FC10084, SCL
TITLE = LGF_Random_DInt
{ S7_Optimized_Access := 'TRUE' }
AUTHOR : Siemens_Digital_Industries
FAMILY : LGF
NAME : LGF_Random_DInt
// Generates a random number in the DInt Range
   VAR_OUTPUT
      error : Bool;   // Error if true
      status : Word;   // Status of the function
      subfunctionStatus : Word;   // Status or return value of called FB's, FCs and system blocks
   END_VAR
   VAR_TEMP
      tempTime : DTL;   // System time
      tempNanoSecondInDWord : DWord;   // UDINT converted to DWORD for access to individual bytes
      tempTimeStatus : Word;   // Status of the instruction RD_SYS_T
      tempRandomValue : DWord;   // Random-start-value
   END_VAR
   // Ret_Val : Random number in the Dint range
   VAR CONSTANT
      ZERO : DInt;   // Zero value in case of error
      SUB_STATUS_NO_ERROR : Word := 16#0000;   // Status: sub function call ends without error
      STATUS_FINISHED_NO_ERROR : Word := 16#0000;   // Status: Execution finished without errors
      ERR_RD_SYS_T : Word := 16#8600;   // Error: System function Read system time returned an error
   END_VAR
BEGIN
   REGION Block info header
     //=============================================================================
     // SIEMENS AG / (c)Copyright 2017
     //-----------------------------------------------------------------------------
     // Title:            LGF_Random_DInt
     // Comment/Function: Generates a random number in the DInt Range
     // Library/Family:   LGF(Library General Functions)
     // Author:           Siemens Digital Industry Support
     // Tested with:      S7-PLCSIM Advanced V2.0 SP1
     // Engineering:      TIA Portal V15 Update 2
     // Restrictions:     ENO disabled - error handling done by error and status
     // Requirements:     PLC (S7-1200 / S7-1500)
     //-------------------------------------------------------------------------------
     // Change log table:
     // Version  | Date       | Expert in charge       | Changes applied
     //----------|------------|------------------------|------------------------------
     // 01.00.00 13.11.2019  Siemens Industry Presales Support
     //                      First release
     //                      copied from "LGF_Random_Real"
     // 03.00.00 23.04.2020  Siemens Industry Support
     //                      Set version to V3.0.0, harmonize the version of the whole library
     //=============================================================================
   END_REGION

   REGION Validation
     // Read system time
     #tempTimeStatus := INT_TO_WORD(RD_SYS_T(#tempTime));

     // Check return variable for error
     IF (#tempTimeStatus <> #SUB_STATUS_NO_ERROR) THEN
       #error := true;
       #status := #ERR_RD_SYS_T;
       #subfunctionStatus := #tempTimeStatus;
       #LGF_Random_DInt := #ZERO;
       RETURN;
     END_IF;
   END_REGION

   REGION Calculating random number
     // Converting to double word so individual bytes can be addressed
     #tempNanoSecondInDWord := UDINT_TO_DWORD(#tempTime.NANOSECOND);

     // Calculate a random-start-value depending on the time
     #tempRandomValue.%B3 := #tempNanoSecondInDWord.%B0;
     #tempRandomValue.%B2 := #tempNanoSecondInDWord.%B1;
     #tempRandomValue.%B1 := #tempNanoSecondInDWord.%B2;
     #tempRandomValue.%B0 := #tempNanoSecondInDWord.%B3;

     #LGF_Random_DInt := DWORD_TO_DINT(#tempRandomValue);

     #error := false;
     #status := #STATUS_FINISHED_NO_ERROR;
     #subfunctionStatus := #SUB_STATUS_NO_ERROR;
     // ENO mechanism is not used
     ENO := TRUE;
   END_REGION
END_FUNCTION